# B&R Automation Studio project 2SegDemo (part 3)

#### WaveParFb.st
```iecst
(*
 This FB only atm works at 1ms cycle time

//Hz is times per second, in this case times is revolutions.
//To convert the Hz to revolutions and then scale by the task class cycle time
//1 hz, would mean that every TC cycle, we'd be incrementing by 2*PI/CycleTime

//Rx and Rz cylcic positions are always relative to the current position at the
//  ENABLING of the cyclic channel. Why? Who knows but that's the way it works
*)
FUNCTION_BLOCK WaveFb
	IF Enable AND Active AND Running THEN
		int.WaveCtrl.WaveX := int.WaveCtrl.WaveX + Pars.Wave.Freq / 1000 * 2 * 3.14;
		int.SlideCtrl.WaveX := int.SlideCtrl.WaveX + Pars.Slide.Freq / 1000 * 2 * 3.14;
		IF int.WaveCtrl.WaveX > 2 * 3.14 THEN
			int.WaveCtrl.WaveX := 0;
		END_IF

		IF int.SlideCtrl.WaveX > 2 * 3.14 THEN
			int.SlideCtrl.WaveX := 0;
		END_IF

		int.WaveCtrl.WaveY := SIN(int.WaveCtrl.WaveX);
		int.WaveCtrl.Height := int.WaveCtrl.WaveY * Pars.Wave.Amp + Pars.Wave.Center;

		//For the angle,just going to scale between -20/+20mRad.
		int.WaveCtrl.Angle := COS(int.WaveCtrl.WaveX) * 20;

		int.SlideCtrl.Height := SIN(int.SlideCtrl.WaveX) * 180 + 240;
	END_IF
	CASE int.State OF
		WAVE_IDLE: //**************************************************************** Idle State
			IF Enable THEN
				int.Fbs.GroupCreateFb.Controller := ADR(Controller);
				int.Fbs.GroupCreateFb.GroupID := 1;
				int.Fbs.GroupCreateFb.NumberOfShuttles := 2;
				int.Fbs.GroupCreateFb.ShuttleID[0] := 1;
				int.Fbs.GroupCreateFb.ShuttleID[1] := 2;
				int.Fbs.GroupCreateFb.Execute := TRUE;

				Active := TRUE;

				int.State := WAVE_CREATE_GROUP;
			END_IF
		WAVE_CREATE_GROUP: //**************************************************************** Create Sh Group
			IF int.Fbs.GroupCreateFb.Error THEN
				int.ErrorState := int.State;
				Error := TRUE;
				int.State := WAVE_ERROR;
			ELSIF int.Fbs.GroupCreateFb.Done THEN
				int.Fbs.GroupCreateFb.Execute := FALSE;

				int.Fbs.GroupCtrlFb.Controller := ADR(Controller);
				int.Fbs.GroupCtrlFb.CoupleMode := mcACP6D_GROUP_COUPLE_ONLY_XY;
				int.Fbs.GroupCtrlFb.GroupID := 1;
				int.Fbs.GroupCtrlFb.Option := mcACP6D_GROUP_COUPLE;
				int.Fbs.GroupCtrlFb.Execute := TRUE;

				int.State := WAVE_BOND_GROUP;
			END_IF
		WAVE_BOND_GROUP: //**************************************************************** Bond Sh Group
			IF int.Fbs.GroupCtrlFb.Error THEN
				int.ErrorState := int.State;
				Error := TRUE;
				int.State := WAVE_ERROR;
			ELSIF int.Fbs.GroupCtrlFb.Done THEN
				int.Fbs.GroupCtrlFb.Execute := FALSE;

				int.Fbs.ShortAxisFb.Controller := ADR(Controller);
				int.Fbs.ShortAxisFb.ShuttleID := 1; //Hard coded to 1 for now
				int.Fbs.ShortAxisFb.PositionZ := (Pars.Wave.Amp + Pars.Wave.Center) / 1000.0;
				int.Fbs.ShortAxisFb.PositionRx := 0.0;
				int.Fbs.ShortAxisFb.PositionRy := 0;
				int.Fbs.ShortAxisFb.PositionRz := 0;
				int.Fbs.ShortAxisFb.VelocityZ := 1;
				int.Fbs.ShortAxisFb.VelocityRx := 1;
				int.Fbs.ShortAxisFb.VelocityRy := 1;
				int.Fbs.ShortAxisFb.VelocityRz := 1;
				int.Fbs.ShortAxisFb.Execute := TRUE;

				int.State := WAVE_CFG_CHANNEL;
			END_IF
		WAVE_CFG_CHANNEL: //**************************************************************** Configure cyclic channel
			IF int.Fbs.ShortAxisFb.Error THEN
				int.ErrorState := int.State;
				Error := TRUE;
				int.State := WAVE_ERROR;
			ELSIF int.Fbs.ShortAxisFb.Done THEN
				int.Fbs.ShortAxisFb.Execute := FALSE;

				//Start at the peak of the sine wave, so pi/2
				int.WaveCtrl.WaveX := 1.57;
				int.SlideCtrl.WaveX := 1.57;
				int.WaveCtrl.WaveY := SIN(int.WaveCtrl.WaveX);
				int.WaveCtrl.Height := int.WaveCtrl.WaveY * Pars.Wave.Amp + Pars.Wave.Center;

				//For the angle,just going to scale between -25/+25mRad.
				int.WaveCtrl.Angle := COS(int.WaveCtrl.WaveX) * 25;

				int.Fbs.CyclicZFb.AxisID := 3;
				int.Fbs.CyclicZFb.ChannelID := 1;
				int.Fbs.CyclicZFb.Controller := ADR(Controller);
				int.Fbs.CyclicZFb.Value := (Pars.Wave.Amp + Pars.Wave.Center) - int.WaveCtrl.Height;
				int.Fbs.CyclicZFb.Enable := TRUE;

				int.Fbs.CyclicRxFb.AxisID := 5;
				int.Fbs.CyclicRxFb.ChannelID := 1;
				int.Fbs.CyclicRxFb.Controller := ADR(Controller);
				int.Fbs.CyclicRxFb.Value := 0;
				int.Fbs.CyclicRxFb.Enable := TRUE;

				int.Fbs.CyclicXFb.AxisID := 1;
				int.Fbs.CyclicXFb.ChannelID := 1;
				int.Fbs.CyclicXFb.Controller := ADR(Controller);
				int.Fbs.CyclicXFb.Value := 0.42;
				int.Fbs.CyclicXFb.Enable := TRUE;
				int.State := WAVE_SET_HEIGHT;
			END_IF

		WAVE_SET_HEIGHT: //**************************************************************** Set the starting height
			int.Fbs.CyclicChCtrlFb.Controller := ADR(Controller);
			int.Fbs.CyclicChCtrlFb.ShuttleID[0] := 1;
			int.Fbs.CyclicChCtrlFb.ChannelID[0] := 1;
			int.Fbs.CyclicChCtrlFb.AxisID[0].0 := TRUE; //X
			int.Fbs.CyclicChCtrlFb.AxisID[0].2 := TRUE; //Z
			int.Fbs.CyclicChCtrlFb.AxisID[0].4 := TRUE; //Ry
			int.Fbs.CyclicChCtrlFb.Execute := TRUE;
			int.Fbs.CyclicChCtrlFb.NumberOfShuttles := 1;
			int.Fbs.CyclicChCtrlFb.Level := 1;

			IF int.Fbs.CyclicChCtrlFb.Error THEN
				int.ErrorState := int.State;
				Error := TRUE;
				int.State := WAVE_ERROR;
			ELSIF int.Fbs.CyclicChCtrlFb.Done THEN
				int.Fbs.CyclicChCtrlFb.Execute := FALSE;
				Running := TRUE;
				int.State := WAVE_WAVE;
			END_IF
		WAVE_WAVE: //**************************************************************** Write channels, ride the wave
			int.Fbs.CyclicZFb.Value := -((Pars.Wave.Amp + Pars.Wave.Center) - int.WaveCtrl.Height) / 1000.0;
			int.Fbs.CyclicRxFb.Value := int.WaveCtrl.Angle / 1000.0;
			int.Fbs.CyclicXFb.Value := int.SlideCtrl.Height / 1000.0;

			IF NOT Enable THEN
				Running := FALSE;
				int.Fbs.CyclicZFb.Enable := FALSE;
				int.Fbs.CyclicRxFb.Enable := FALSE;
				int.Fbs.CyclicXFb.Enable := FALSE;
				int.Fbs.CyclicChCtrlFb.Execute := TRUE;
				int.Fbs.CyclicChCtrlFb.Level := 0;

				int.State := WAVE_EXIT_CFG;
			END_IF
		WAVE_EXIT_CFG:  //**************************************************************** Exit config channel
			IF int.Fbs.CyclicChCtrlFb.Error THEN
				int.ErrorState := int.State;
				Error := TRUE;
				int.State := WAVE_ERROR;
			ELSIF int.Fbs.CyclicChCtrlFb.Done THEN
				int.Fbs.CyclicChCtrlFb.Execute := FALSE;

				int.Fbs.ShortAxisFb.Controller := ADR(Controller);
				int.Fbs.ShortAxisFb.ShuttleID := 1;
				int.Fbs.ShortAxisFb.PositionZ := Pars.DefaultLevitationHeight;
				int.Fbs.ShortAxisFb.PositionRx := 0.0;
				int.Fbs.ShortAxisFb.PositionRy := 0;
				int.Fbs.ShortAxisFb.PositionRz := 0;
				int.Fbs.ShortAxisFb.VelocityZ := 1;
				int.Fbs.ShortAxisFb.VelocityRx := 1;
				int.Fbs.ShortAxisFb.VelocityRy := 1;
				int.Fbs.ShortAxisFb.VelocityRz := 1;
				int.Fbs.ShortAxisFb.Execute := TRUE;

				int.State := WAVE_MOVE_BACK;
			END_IF
		WAVE_MOVE_BACK: //**************************************************************** Move Back to level
			IF int.Fbs.ShortAxisFb.Error THEN
				int.ErrorState := int.State;
				Error := TRUE;
				int.State := WAVE_ERROR;
			ELSIF int.Fbs.ShortAxisFb.Done THEN
				int.Fbs.ShortAxisFb.Execute := FALSE;

				int.Fbs.GroupCtrlFb.Option := mcACP6D_GROUP_DECOUPLE;
				int.Fbs.GroupCtrlFb.Execute := TRUE;

				int.State := WAVE_UNBOUND_GROUP;
			END_IF
		WAVE_UNBOUND_GROUP: //**************************************************************** Unbond Sh Group
			IF int.Fbs.GroupCtrlFb.Error THEN
				int.ErrorState := int.State;
				Error := TRUE;
				int.State := WAVE_ERROR;
			ELSIF int.Fbs.GroupCtrlFb.Done THEN
				int.Fbs.GroupCtrlFb.Execute := FALSE;

				int.Fbs.GroupDeleteFb.Controller := ADR(Controller);
				int.Fbs.GroupDeleteFb.GroupID := 1;
				int.Fbs.GroupDeleteFb.Execute := TRUE;

				int.State := WAVE_DELETE_GROUP;
			END_IF
		WAVE_DELETE_GROUP: //**************************************************************** Delete Sh Group
			IF int.Fbs.GroupDeleteFb.Error THEN
				int.ErrorState := int.State;
				Error := TRUE;
				int.State := WAVE_ERROR;
			ELSIF int.Fbs.GroupDeleteFb.Done THEN
				int.Fbs.GroupDeleteFb.Execute := FALSE;

				Active := FALSE;
				int.WaveCtrl.WaveX := 0;
				int.SlideCtrl.WaveX := 0;
				int.State := WAVE_IDLE;
			END_IF
		WAVE_ERROR: //**************************************************************** Error State
			IF NOT Enable THEN

				Active := FALSE;
				Error := FALSE;
				Running := FALSE;

				int.Fbs.ShortAxisFb.Execute := FALSE;
				int.Fbs.CyclicChCtrlFb.Execute := FALSE;
				int.Fbs.CyclicZFb.Enable := FALSE;
				int.Fbs.CyclicRxFb.Enable := FALSE;
				int.Fbs.CyclicXFb.Enable := FALSE;
				int.Fbs.GroupCreateFb.Execute := FALSE;
				int.Fbs.GroupCtrlFb.Execute := FALSE;
				int.Fbs.GroupDeleteFb.Execute := FALSE;

				int.WaveCtrl.WaveX := 0;
				int.SlideCtrl.WaveX := 0;
				int.State := WAVE_IDLE;
			END_IF

	END_CASE;

	int.Fbs.ShortAxisFb();
	int.Fbs.CyclicChCtrlFb();
	int.Fbs.CyclicZFb();
	int.Fbs.CyclicRxFb();
	int.Fbs.CyclicXFb();
	int.Fbs.GroupCreateFb();
	int.Fbs.GroupCtrlFb();
	int.Fbs.GroupDeleteFb();

END_FUNCTION_BLOCK
```

#### AntiSloshFb.st
```iecst
FUNCTION_BLOCK AntiSloshFb

END_FUNCTION_BLOCK
```

#### LandFb.st
```iecst
FUNCTION_BLOCK LandFb

	CASE int.State OF
		LAND_IDLE: //**************************************************************** Idle State
			IF Enable THEN
				Active := TRUE;

				int.State := LAND_WAIT;
			END_IF
		LAND_ISSUE_CMD: //**************************************************************** Create Sh Group
			IF int.Fbs.LandFb.Error THEN
				int.ErrorState := int.State;
				Error := TRUE;
				int.State := LAND_ERROR;
			ELSIF NOT Enable AND int.Fbs.LandFb.Done THEN
				int.Fbs.LandFb.Execute := FALSE;

				int.State := LAND_RESET;
			ELSIF int.Fbs.LandFb.Done THEN
				int.Landed := NOT int.Landed;
				int.Fbs.LandFb.Execute := FALSE;

				int.State := LAND_WAIT;
			END_IF
		LAND_WAIT: //**************************************************************** Waiting for an update cmd
			IF NOT Enable THEN
				IF Land THEN
					int.Fbs.LandFb.Controller := ADR(Controller);
					int.Fbs.LandFb.Level := mcACP6D_LEVEL_LEVITATE;
					int.Fbs.LandFb.ShuttleID := Pars.ShId;
					int.Fbs.LandFb.Execute := TRUE;

					int.State := LAND_ISSUE_CMD;
				ELSE
					int.State := LAND_RESET;
				END_IF
			ELSIF (Land AND NOT int.Landed) OR (NOT Land AND int.Landed) THEN
				IF int.Landed THEN
					int.Fbs.LandFb.Level := mcACP6D_LEVEL_LEVITATE;
				ELSE
					int.Fbs.LandFb.Level := mcACP6D_LEVEL_LAND;
				END_IF
				int.Fbs.LandFb.Controller := ADR(Controller);
				int.Fbs.LandFb.ShuttleID := Pars.ShId;
				int.Fbs.LandFb.Execute := TRUE;

				int.State := LAND_ISSUE_CMD;
			END_IF

		LAND_ERROR: //**************************************************************** Error STate
			IF NOT Enable THEN
				int.State := LAND_RESET;
			END_IF

		LAND_RESET: //**************************************************************** Reset state
			Active := FALSE;
			Error := FALSE;
			int.Landed := FALSE;

			int.Fbs.LandFb.Execute := FALSE;

			int.State := LAND_IDLE;
	END_CASE;

	int.Fbs.LandFb();
END_FUNCTION_BLOCK
```

#### GenericDemoFb.st
```iecst
FUNCTION_BLOCK GenericMotionDemoFB

	CASE int.State OF
		GEN_IDLE: //**************************************************************** Idle State
			IF Enable THEN
				Active := TRUE;

				int.Fbs.BufferCtrl.Controller := ADR(Controller);
				int.Fbs.BufferCtrl.Option := mcACP6D_BUFFER_BLOCK;
				int.Fbs.BufferCtrl.ShuttleID := 0;
				int.Fbs.BufferCtrl.Execute := TRUE;

				int.State := GEN_BLOCK_BUFFER;
			END_IF
		GEN_BLOCK_BUFFER: //**************************************************************** Block Buffer
			IF int.Fbs.BufferCtrl.Error THEN
				int.ErrorState := int.State;
				Error := TRUE;
				int.State := GEN_ERROR;
			ELSIF int.Fbs.BufferCtrl.Done THEN
				int.Fbs.BufferCtrl.Execute := FALSE;

				int.Fbs.MacroRunFB.Controller := ADR(Controller);
				int.Fbs.MacroRunFB.ShuttleID := Pars.ShId[0];
				int.Fbs.MacroRunFB.MacroID := Pars.MacroId[0];
				int.Fbs.MacroRunFB.Execute := TRUE;

				int.State := GEN_RUN_MACRO1;
			END_IF
		GEN_RUN_MACRO1: //**************************************************************** Run Macro 1
			IF int.Fbs.MacroRunFB.Error THEN
				int.ErrorState := int.State;
				Error := TRUE;
				int.State := GEN_ERROR;
			ELSIF int.Fbs.MacroRunFB.Acknowledge THEN
				int.Fbs.MacroRunFB.Execute := FALSE;
				int.Fbs.MacroRunFB.ShuttleID := Pars.ShId[1];
				int.Fbs.MacroRunFB.MacroID := Pars.MacroId[1];

				int.State := GEN_RUN_MACRO2;
			END_IF
		GEN_RUN_MACRO2: //**************************************************************** Run Macro 2
			int.Fbs.MacroRunFB.Execute := TRUE;
			IF int.Fbs.MacroRunFB.Error THEN
				int.ErrorState := int.State;
				Error := TRUE;
				int.State := GEN_ERROR;
			ELSIF int.Fbs.MacroRunFB.Acknowledge THEN
				int.Fbs.MacroRunFB.Execute := FALSE;

				int.Fbs.BufferCtrl.Option := mcACP6D_BUFFER_RELEASE;
				int.Fbs.BufferCtrl.Execute := TRUE;

				int.State := GEN_RELEASE_BUFFER;
			END_IF

		GEN_RELEASE_BUFFER: //**************************************************************** Block Buffer
			IF int.Fbs.BufferCtrl.Error THEN
				int.ErrorState := int.State;
				Error := TRUE;
				int.State := GEN_ERROR;
			ELSIF int.Fbs.BufferCtrl.Done THEN
				int.Fbs.BufferCtrl.Execute := FALSE;

				int.State := GEN_RUN_DEMO;
			END_IF
		GEN_RUN_DEMO: //**************************************************************** Run Demo State
			IF NOT Enable THEN
				int.Fbs.StopFb.Controller := ADR(Controller);
				int.Fbs.StopFb.ShuttleID := 0;
				int.Fbs.StopFb.Execute := TRUE;
				int.State := GEN_STOP;
			END_IF
		GEN_STOP:  //**************************************************************** Stopping Shuttle state
			IF int.Fbs.StopFb.Error THEN
				int.ErrorState := int.State;
				Error := TRUE;
				int.State := GEN_ERROR;
			ELSIF int.Fbs.StopFb.Done THEN
				int.Fbs.StopFb.Execute := FALSE;

				int.Fbs.ShortAxisFb.Controller := ADR(Controller);
				int.Fbs.ShortAxisFb.PositionZ := 0.001;
				int.Fbs.ShortAxisFb.ShuttleID := Pars.ShId[0];
				int.Fbs.ShortAxisFb.VelocityZ := 1;
				int.Fbs.ShortAxisFb.Execute := TRUE;

				int.State := GEN_RESET_HEIGHT1;
			END_IF
		GEN_RESET_HEIGHT1: //**************************************************************** Reset Height 1
			IF int.Fbs.ShortAxisFb.Error THEN
				int.ErrorState := int.State;
				Error := TRUE;
				int.State := GEN_ERROR;
			ELSIF int.Fbs.ShortAxisFb.Done THEN
				int.Fbs.ShortAxisFb.Execute := FALSE;

				int.Fbs.ShortAxisFb.ShuttleID := Pars.ShId[1];
				int.State := GEN_RESET_HEIGHT2;
			END_IF
		GEN_RESET_HEIGHT2: //**************************************************************** Reset Height 2
			int.Fbs.ShortAxisFb.Execute := TRUE;
			IF int.Fbs.ShortAxisFb.Error THEN
				int.ErrorState := int.State;
				Error := TRUE;
				int.State := GEN_ERROR;
			ELSIF int.Fbs.ShortAxisFb.Done THEN
				int.Fbs.ShortAxisFb.Execute := FALSE;

				int.State := GEN_RESET;
			END_IF
		GEN_ERROR: //**************************************************************** Error state
			IF NOT Enable THEN
				int.State := GEN_RESET;
			END_IF

		GEN_RESET: //**************************************************************** Reset state
			Active := FALSE;
			Error := FALSE;

			int.Fbs.ShortAxisFb.Execute := FALSE;
			int.Fbs.BufferCtrl.Execute := FALSE;
			int.Fbs.MacroRunFB.Execute := FALSE;
			int.Fbs.StopFb.Execute := FALSE;

			int.State := GEN_IDLE;;
	END_CASE;

	int.Fbs.ShortAxisFb();
	int.Fbs.BufferCtrl();
	int.Fbs.MacroRunFB();
	int.Fbs.StopFb();

END_FUNCTION_BLOCK
```

### Program Logical/Source/Demos/MixDemo

#### Types.typ
```iecst
TYPE
	MoveTyp : 	STRUCT
		X : REAL;
		Y : REAL;
		Vel : REAL;
		Accel : REAL;
		EndVel : REAL;
		Angle : REAL;
	END_STRUCT;
	FbsTyp : 	STRUCT
		MovePlaneFb : MC_BR_MoveInPlane_Acp6D;
		MoveArcFb : MC_BR_MoveArcAngle_Acp6D;
		Wait : TON;
		RunMacroFb : MC_BR_MacroRun_Acp6D;
		LoadMacroFb : MC_BR_MacroLoad_Acp6D;
	END_STRUCT;
END_TYPE
```

#### Variables.var
```iecst
VAR
	Fbs : FbsTyp;
	state : UDINT;
	shId : USINT;
END_VAR
VAR RETAIN
	run : BOOL;
END_VAR
VAR
	macroId : USINT;
END_VAR
```

#### Cyclic.st
```iecst
//Mixing demo

(*
	Move shuttle to segment center position
	Wait for some time (here food coloring is added)
	Preform mixing movement
	Move back to other side
	Wait for some time (food coloring added)
	Preform mixing movement
	Move shuttle to start position

*)

PROGRAM _CYCLIC
	Fbs.LoadMacroFb.Controller := ADR(gMcAcp6DController);

	Fbs.RunMacroFb.Controller := ADR(gMcAcp6DController);
	Fbs.RunMacroFb.ShuttleID := shId;
	Fbs.RunMacroFb.MacroID := macroId;

	CASE state OF
		0:
			Fbs.LoadMacroFb.MacroID := macroId;
			IF run THEN
				Fbs.RunMacroFb.Execute := TRUE;
				Fbs.RunMacroFb.MacroID := 130;
				state := 10;
			END_IF
		10:
			IF Fbs.RunMacroFb.Done THEN
				Fbs.RunMacroFb.Execute := FALSE;
				state := 11;
			END_IF
		11:
			Fbs.RunMacroFb.Execute := TRUE;
			Fbs.RunMacroFb.MacroID := 131;
			state := 20;
		20:
			IF Fbs.RunMacroFb.Done THEN
				Fbs.RunMacroFb.Execute := FALSE;
				state := 21;
			END_IF
		21:
			Fbs.RunMacroFb.Execute := TRUE;
			Fbs.RunMacroFb.MacroID := 132;
			state := 30;
		30:
			IF Fbs.RunMacroFb.Done THEN
				Fbs.RunMacroFb.Execute := FALSE;
				state := 31;
			END_IF
		31:
			Fbs.RunMacroFb.Execute := TRUE;
			Fbs.RunMacroFb.MacroID := 131;
			state := 40;
		40:
			IF Fbs.RunMacroFb.Done THEN
				Fbs.RunMacroFb.Execute := FALSE;

				Fbs.MovePlaneFb.Controller := ADR(gMcAcp6DController);
				Fbs.MovePlaneFb.ShuttleID := shId;
				Fbs.MovePlaneFb.PositionX := 0.24;
				Fbs.MovePlaneFb.PositionY := 0.12;
				Fbs.MovePlaneFb.Velocity := 0.5;
				Fbs.MovePlaneFb.Acceleration := 1;
				Fbs.MovePlaneFb.Execute := TRUE;
				state := 50;
			END_IF
		50:
			IF Fbs.MovePlaneFb.Done THEN
				Fbs.MovePlaneFb.Execute := FALSE;
				run := FALSE;
				state := 0;
			END_IF
	END_CASE;

	Fbs.LoadMacroFb();
	Fbs.MovePlaneFb();
	Fbs.RunMacroFb();
END_PROGRAM
```

#### Init.st
```iecst
PROGRAM _INIT
	Fbs.LoadMacroFb.FileDevice := '6DMacro';
	Fbs.LoadMacroFb.FileName := '130_MixDemo.xml';
	macroId := 130;
	shId := 1;
END_PROGRAM
```

### Package Logical/Source/Main - Package that contains the main entry point to the machine

### Program Logical/Source/Main/Main

#### Types.typ
```iecst
TYPE
	MainFbsTyp : 	STRUCT
		TimerFb : TON;
		StopAllFb : MC_BR_Stop_Acp6D;
	END_STRUCT;
	MainStatesEnum :
		(
		MAIN_OFF,
		MAIN_INIT,
		MAIN_RECOVERING,
		MAIN_READY,
		MAIN_STARTING,
		MAIN_RUN_PROCESS,
		MAIN_RUN_DANCE,
		MAIN_STOPPING,
		MAIN_ERROR,
		MAIN_RESET
		);
END_TYPE
```

#### Variables.var
```iecst
VAR
	i : USINT; (*Loop index*)
	state : MainStatesEnum; (*State of system*)
	Fbs : MainFbsTyp;
END_VAR
```

#### Cyclic.st
```iecst
PROGRAM _CYCLIC
	IF gAcp6DCtrlIf.Sts.Error THEN
		state := MAIN_ERROR;
	END_IF

	IF gMainIf.Cmd.StopAllShuttles THEN
		Fbs.StopAllFb.Controller := ADR(gMcAcp6DController);
		Fbs.StopAllFb.Execute := TRUE;
		IF Fbs.StopAllFb.Done OR Fbs.StopAllFb.Error THEN
			Fbs.StopAllFb.Execute := FALSE;
			gMainIf.Cmd.StopAllShuttles := FALSE;
		END_IF
	END_IF

	CASE state OF
		MAIN_OFF: //******************************************************************************** Main Off State
			IF gMainIf.Cmd.Power THEN
				gAcp6DCtrlIf.Cmd.Power := gMainIf.Cfg.Enable6D;

				state := MAIN_INIT;
			END_IF

		MAIN_INIT: //******************************************************************************** Main Initializing State
			IF (gAcp6DCtrlIf.Sts.PowerOn AND gAcp6DCtrlIf.Sts.Ready OR NOT gMainIf.Cfg.Enable6D) THEN
				gMainIf.Sts.Power6D := TRUE;

				state := MAIN_READY;
			ELSIF NOT gMainIf.Cmd.Power THEN
				gAcp6DCtrlIf.Cmd.Power := FALSE;

				gMainIf.Sts.Power6D := FALSE;

				state := MAIN_OFF;
			END_IF
		MAIN_RECOVERING: //******************************************************************************** Main Recovery State
			IF (g6DRecoveryIf.Sts.ReadyToStartProc OR NOT gMainIf.Cfg.Enable6D) THEN
				g6DRecoveryIf.Cmd.Recover := FALSE;

				state := MAIN_READY;
			END_IF
		MAIN_READY://******************************************************************************** Main Ready State
			IF NOT gMainIf.Cmd.Power THEN
				gMainIf.Sts.Power6D := FALSE;
				gAcp6DCtrlIf.Cmd.Power := FALSE;

				state := MAIN_OFF;
			END_IF

		MAIN_STARTING://******************************************************************************** Main Starting State
			IF gAcp6DCtrlIf.Sts.Error THEN
				state := MAIN_ERROR;
			ELSIF NOT gMainIf.Cmd.Power THEN
				gMainIf.Cmd.StartDemoCycle := FALSE;
				gMainIf.Sts.Power6D := FALSE;
				gAcp6DCtrlIf.Cmd.Power := FALSE;

				state := MAIN_OFF;
			END_IF

		MAIN_RUN_PROCESS: //******************************************************************************** Main Process State
		MAIN_STOPPING: //******************************************************************************** Main Stopping State

		MAIN_ERROR: //******************************************************************************** Main Error State
			IF gMainIf.Cmd.Reset THEN
				gMainIf.Cmd.Reset := FALSE;

				gMainIf.Sts.Running := FALSE;
				gAcp6DCtrlIf.Cmd.ErrorReset := TRUE;
				Fbs.TimerFb.IN := FALSE;

				IF gMainIf.Cmd.Power THEN
					state := MAIN_READY;
				ELSE
					state := MAIN_OFF;
				END_IF
			END_IF
	END_CASE;

	Fbs.StopAllFb();
END_PROGRAM
```

#### Init.st
```iecst
PROGRAM _INIT
	gMainIf.Cfg.ShuttleCount := 8;

	gMainIf.Cfg.Enable6D := TRUE;
	gMainIf.Cfg.EnableRobot := TRUE;

	gMainIf.Par.ProcessDemoTime := T#120s;
	gMainIf.Par.DanceDemoTime := T#180s;

	//Used to initialize the shuttle indecies.
	FOR i:=0 TO gMainIf.Cfg.ShuttleCount-1 DO
		gShuttleIf[i].Cfg.ShuttleId := i + 1;
	END_FOR;

END_PROGRAM
```

### Package Logical/Source/6DCtrl - Package containing the main logic for controlling the 6D system as a whole

### Acp6DTypes.typ
```iecst
(*Datatypes for the Load Macro Interface*)

TYPE
	gMacroLoadIfTYp : 	STRUCT
		Cmd : gMacroLoadIfCmdTyp;
		Par : gMacroLoadIfParTyp;
		Sts : gMacroLoadIfStatusTyp;
	END_STRUCT;
	gMacroLoadIfCmdTyp : 	STRUCT
		LoadAll : BOOL; (*Command to load all macros*)
		Clear : BOOL; (*Command to clear a singular macro*)
		LoadSingle : BOOL; (*Commadn to load a singular macro*)
		Reset : BOOL; (*Command to reset the macro load interface. Also resets the "AllMacroLoaded" status*)
	END_STRUCT;
	MacroParTyp : 	STRUCT
		Load : BOOL; (*Flag To denote that we should load the macro*)
		MacroFileName : STRING[80]; (*XML File Name of the Macro to load*)
		MacroID : USINT; (*MacroID of the associated macro*)
	END_STRUCT;
	gMacroLoadIfParTyp : 	STRUCT
		FileDevice : STRING[80]; (*FileDevice to find the macro *)
		MacroList : ARRAY[0..MAX_MACRO_COUNT_ARRAY]OF MacroParTyp; (*List of macros to load*)
		SingleMacroLoad : MacroParTyp; (*Parameter to load a singular macro*)
	END_STRUCT;
	gMacroLoadIfStatusTyp : 	STRUCT
		AllMacrosLoaded : BOOL;
		Loading : BOOL;
		CurrentMacro : USINT;
		CmdDone : BOOL;
		Error : BOOL;
		MacroIDError : USINT;
	END_STRUCT;
END_TYPE
```

### Program Logical/Source/6DCtrl/6DCtrl (IEC)

#### Cyclic.st
```iecst
PROGRAM _CYCLIC

	IF((Fbs.SysReadStateFb.Valid AND Fbs.SysReadStateFb.State = mcACP6D_STATE_ERROR) AND (state <> ACP6D_ERROR))THEN
		state := ACP6D_ERROR;
	END_IF;

	CASE state OF
		ACP6D_RESET: 	//******************************************************************************** 6D Reset State
			IF(Fbs.SysReadStateFb.Valid AND (Fbs.SysReadStateFb.State = mcACP6D_STATE_INACTIVE))THEN
				state := ACP6D_INACTIVE;
			ELSIF(Fbs.SysReadStateFb.State = mcACP6D_STATE_OPERATION)THEN
				state := ACP6D_POWER_OFF;
			END_IF;

		ACP6D_POWER_OFF: 	//******************************************************************************** 6D Power off commanding State
			Fbs.PowerOffFb.Execute := TRUE;
			IF(Fbs.PowerOffFb.Acknowledge AND (Fbs.SysReadStateFb.Valid AND Fbs.SysReadStateFb.State = mcACP6D_STATE_INACTIVE))THEN
				gAcp6DCtrlIf.Sts.PowerOn := FALSE;
				Fbs.PowerOffFb.Execute 	:= FALSE;
				state := ACP6D_INACTIVE;
			ELSIF(Fbs.PowerOffFb.Error)THEN
				Fbs.PowerOffFb.Execute 	:= FALSE;
				gAcp6DCtrlIf.Sts.ErrorID := Fbs.PowerOffFb.ErrorID;
				state := ACP6D_ERROR;
			END_IF;

		ACP6D_INACTIVE:	 	//******************************************************************************** 6D Inactive/Power Off state
			IF(gAcp6DCtrlIf.Cmd.Power)THEN
				Fbs.PowerOnFb.Execute := TRUE;
				//MpAuditCustomEvent(gAuditTrail,"INFO","Acp6DSys","Power On Command Issued");
				state := ACP6D_POWER_ON;
			END_IF;

		ACP6D_POWER_ON: 	//******************************************************************************** 6D Power on Commanding State
			IF Fbs.PowerOnFb.Error THEN
				gAcp6DCtrlIf.Sts.ErrorID := Fbs.PowerOnFb.ErrorID;
				state := ACP6D_ERROR;
			ELSIF(Fbs.PowerOnFb.Acknowledge AND (Fbs.SysReadStateFb.Valid AND (Fbs.SysReadStateFb.State > mcACP6D_STATE_INACTIVE)))THEN
				//MpAuditCustomEvent(gAuditTrail,"INFO","Acp6DSys","Powered On");
				Fbs.PowerOnFb.Execute := FALSE;
				state := ACP6D_WAIT_ACTIVATION;
			END_IF;

			//Necessary state when using Absolute ID.
		ACP6D_WAIT_ACTIVATION: 	//******************************************************************************** 6D Waiting for Activation of Shuttles State
			IF(Fbs.SysReadStateFb.Valid)THEN
				IF(Fbs.SysReadStateFb.State = mcACP6D_STATE_OPERATION)THEN
					gAcp6DCtrlIf.Sts.PowerOn := TRUE;
					IF gAcp6DCtrlIf.Par.MacroEnabled THEN

						state := ACP6D_INIT_MACRO;
					ELSE
						state := ACP6D_READY;
					END_IF
				ELSIF(Fbs.SysReadStateFb.State = mcACP6D_STATE_INACTIVE)THEN
					state := ACP6D_INACTIVE; // Error during Activating state; Can happen in Absolute ID mode.
					gAcp6DCtrlIf.Cmd.Power := FALSE;
				END_IF;
			END_IF;
		ACP6D_INIT_MACRO: 	//******************************************************************************** 6D Wait for Macro initilization State
			IF gMacroLoadIf.Sts.AllMacrosLoaded THEN
				gMacroLoadIf.Cmd.LoadAll := FALSE;

				state := ACP6D_READY;
			ELSE
				gMacroLoadIf.Cmd.LoadAll := TRUE;
			END_IF
		ACP6D_CFG_CYCLIC_CHANNEL: 	//******************************************************************************** 6D Confiugring the cyclic channel reads
			IF Fbs.CfgReadCyclicPos.Error THEN
				gAcp6DCtrlIf.Sts.Error := TRUE;
				gAcp6DCtrlIf.Sts.ErrorID := Fbs.CfgReadCyclicPos.ErrorID;

				state := ACP6D_ERROR;
			ELSIF Fbs.CfgReadCyclicPos.Done THEN
				Fbs.CfgReadCyclicPos.Execute := FALSE;

				state := ACP6D_READY;
			END_IF
		ACP6D_READY: 	//******************************************************************************** 6D Ready/Running State
			IF(NOT gAcp6DCtrlIf.Cmd.Power)THEN
				gMacroLoadIf.Cmd.Reset := TRUE;
				state := ACP6D_POWER_OFF;
			END_IF;

		ACP6D_ERROR: 	//******************************************************************************** 6D Error State
			gAcp6DCtrlIf.Sts.PowerOn := FALSE;
			IF(gAcp6DCtrlIf.Cmd.ErrorReset)THEN
				IF(Fbs.SysReadStateFb.State<>mcACP6D_STATE_ERROR)THEN
					gAcp6DCtrlIf.Cmd.ErrorReset := FALSE;
					state := ACP6D_RESET;
				ELSE
					Fbs.PowerOffFb.Execute := TRUE;	 // Reset error with power off.
					IF(Fbs.PowerOffFb.Acknowledge)THEN
						gMacroLoadIf.Cmd.Reset := TRUE;
						Fbs.PowerOffFb.Execute 	:= FALSE;
					ELSIF(Fbs.PowerOffFb.Error)THEN
						gAcp6DCtrlIf.Cmd.ErrorReset := FALSE;
						Fbs.PowerOffFb.Execute 	:= FALSE;
						gAcp6DCtrlIf.Sts.ErrorID := Fbs.PowerOffFb.ErrorID;
						state := ACP6D_ERROR;
					END_IF;
				END_IF;
			END_IF;
	END_CASE;

	FOR i:=0 TO gMainIf.Cfg.ShuttleCount - 1 DO
		Fbs.ShReadPositionFb[i].Controller := ADR(gMcAcp6DController);
		Fbs.ShReadPositionFb[i].Enable := TRUE;
		Fbs.ShReadPositionFb[i].ShuttleID := gShuttleIf[i].Cfg.ShuttleId;
		Fbs.ShReadPositionFb[i]();

		Fbs.ShReadForceFb[i].Controller := ADR(gMcAcp6DController);
		Fbs.ShReadForceFb[i].Enable := TRUE;
		Fbs.ShReadForceFb[i].ShuttleID := gShuttleIf[i].Cfg.ShuttleId;
		Fbs.ShReadForceFb[i]();

		Fbs.ShReadState[i].Controller := ADR(gMcAcp6DController);
		Fbs.ShReadState[i].Enable := TRUE;
		Fbs.ShReadState[i].ShuttleID := gShuttleIf[i].Cfg.ShuttleId;
		Fbs.ShReadState[i]();

		gShuttleIf[i].Sts.ShuttleInfo.Force.Value := Fbs.ShReadForceFb[i].ForceInfo;
		gShuttleIf[i].Sts.ShuttleInfo.Force.Valid := Fbs.ShReadForceFb[i].Valid;
		gShuttleIf[i].Sts.ShuttleInfo.Position.Value := Fbs.ShReadPositionFb[i].PositionInfo;
		gShuttleIf[i].Sts.ShuttleInfo.Position.Valid := Fbs.ShReadPositionFb[i].Valid;
		gShuttleIf[i].Sts.ShuttleInfo.State.Value := Fbs.ShReadState[i].State;
		gShuttleIf[i].Sts.ShuttleInfo.State.Valid := Fbs.ShReadState[i].Valid;
	END_FOR;

	IF gAcp6DCtrlIf.Cmd.GetErrorInfo THEN
		Fbs.GetErrorCodesFb.Controller := ADR(gMcAcp6DController);
		Fbs.GetErrorCodesFb.Execute := TRUE;

		IF Fbs.GetErrorCodesFb.Valid OR Fbs.GetErrorCodesFb.Error THEN
			gAcp6DCtrlIf.Sts.ErrorCodes := Fbs.GetErrorCodesFb.ErrorCodes;
			Fbs.GetErrorCodesFb.Execute := FALSE;
			gAcp6DCtrlIf.Cmd.GetErrorInfo := FALSE;
		END_IF

	END_IF
	Fbs.CfgReadCyclicPos();
	Fbs.GetErrorCodesFb();
	Fbs.SysReadStateFb();
	Fbs.PowerOffFb();
	Fbs.PowerOnFb();
	Fbs.AutoRefreshFB();

	gAcp6DCtrlIf.Sts.Ready := state = ACP6D_READY;
	gAcp6DCtrlIf.Sts.Error := state = ACP6D_ERROR;
	gAcp6DCtrlIf.Sts.ReadyToPowerOn := Fbs.SysReadStateFb.Valid AND Fbs.SysReadStateFb.State = mcACP6D_STATE_INACTIVE;
END_PROGRAM
```

#### Init.st
```iecst
PROGRAM _INIT
	gMcAcp6DController.H2P_START := ADR(FBout);
	gMcAcp6DController.P2H_START := ADR(FBin);
	gMcAcp6DController.ConfiguredFeedbackStreamAxis	:= 63;

	Fbs.AutoRefreshFB.Controller	:= ADR(gMcAcp6DController);
	Fbs.PowerOffFb.Controller := ADR(gMcAcp6DController);
	Fbs.PowerOnFb.Controller := ADR(gMcAcp6DController);
	Fbs.SysReadStateFb.Controller := ADR(gMcAcp6DController);

	Fbs.AutoRefreshFB.Enable := TRUE;
	Fbs.SysReadStateFb.Enable := TRUE;

	gAcp6DCtrlIf.Par.MacroEnabled := TRUE;
END_PROGRAM
```

### Program Logical/Source/6DCtrl/MacroLoad (IEC)

#### Cyclic.st
```iecst
PROGRAM _CYCLIC
	CASE state OF
		MACLOAD_IDLE:	//******************************************************************************** Macro Idle State
			IF gMacroLoadIf.Cmd.LoadAll OR gMacroLoadIf.Cmd.LoadSingle THEN
				gMacroLoadIf.Sts.AllMacrosLoaded := FALSE;
				gMacroLoadIf.Sts.Loading := TRUE;
				gMacroLoadIf.Sts.CurrentMacro := 0;

				state := MACLOAD_COUNT_CHECK;
			ELSIF gMacroLoadIf.Cmd.Clear THEN
				MacroFbs.MacroClearFb.Controller := ADR(gMcAcp6DController);
				MacroFbs.MacroClearFb.MacroID := gMacroLoadIf.Par.SingleMacroLoad.MacroID;
				MacroFbs.MacroClearFb.Execute := TRUE;

				state := MACLOAD_CLEAR;
			ELSIF gMacroLoadIf.Cmd.Reset THEN
				gMacroLoadIf.Sts.AllMacrosLoaded := FALSE;
				gMacroLoadIf.Cmd.Reset := FALSE;
			END_IF

		MACLOAD_LOAD://******************************************************************************** Macro Load State
			IF MacroFbs.MacroLoadFb.Error THEN
				gMacroLoadIf.Sts.Error := TRUE;
				gMacroLoadIf.Sts.MacroIDError := gMacroLoadIf.Sts.CurrentMacro;

				state := MACLOAD_ERROR;
			ELSIF MacroFbs.MacroLoadFb.Done THEN
				MacroFbs.MacroLoadFb.Execute := FALSE;
				IF gMacroLoadIf.Cmd.LoadSingle THEN
					gMacroLoadIf.Cmd.LoadSingle := FALSE;
					gMacroLoadIf.Sts.CmdDone := TRUE;
					state := MACLOAD_DONE;
				ELSE //Means we commanded a "LOAD ALL"
					gMacroLoadIf.Sts.CurrentMacro := gMacroLoadIf.Sts.CurrentMacro + 1;

					state := MACLOAD_COUNT_CHECK;
				END_IF
			END_IF

		MACLOAD_COUNT_CHECK: //******************************************************************************** Macro Count check State
			IF gMacroLoadIf.Par.MacroList[gMacroLoadIf.Sts.CurrentMacro].Load THEN
				MacroFbs.MacroLoadFb.Controller := ADR(gMcAcp6DController);
				MacroFbs.MacroLoadFb.FileDevice := gMacroLoadIf.Par.FileDevice;
				IF gMacroLoadIf.Cmd.LoadAll THEN
					MacroFbs.MacroLoadFb.MacroID := gMacroLoadIf.Par.MacroList[gMacroLoadIf.Sts.CurrentMacro].MacroID;
					MacroFbs.MacroLoadFb.FileName := gMacroLoadIf.Par.MacroList[gMacroLoadIf.Sts.CurrentMacro].MacroFileName;

				ELSIF gMacroLoadIf.Cmd.LoadSingle THEN
					MacroFbs.MacroLoadFb.MacroID := gMacroLoadIf.Par.SingleMacroLoad.MacroID;
					MacroFbs.MacroLoadFb.FileName := gMacroLoadIf.Par.SingleMacroLoad.MacroFileName;
				END_IF
				MacroFbs.MacroLoadFb.Execute := TRUE;
				state := MACLOAD_LOAD;
			ELSE
				gMacroLoadIf.Sts.CurrentMacro := gMacroLoadIf.Sts.CurrentMacro + 1;
				IF gMacroLoadIf.Sts.CurrentMacro >= MAX_MACRO_COUNT THEN
					gMacroLoadIf.Sts.AllMacrosLoaded := TRUE;
					gMacroLoadIf.Sts.CmdDone := TRUE;

					state := MACLOAD_DONE;
				END_IF
			END_IF
		MACLOAD_CLEAR: //******************************************************************************** Macro Clear state
			IF MacroFbs.MacroClearFb.Error THEN
				gMacroLoadIf.Sts.Error := TRUE;

				state := MACLOAD_ERROR;
			ELSIF MacroFbs.MacroClearFb.Done THEN
				MacroFbs.MacroClearFb.Execute := FALSE;
				gMacroLoadIf.Sts.CmdDone := TRUE;

				state := MACLOAD_DONE;
			END_IF
		MACLOAD_DONE: //******************************************************************************** Load Done State
			gMacroLoadIf.Sts.Loading := FALSE;
			IF NOT gMacroLoadIf.Cmd.Clear AND NOT gMacroLoadIf.Cmd.LoadAll AND NOT gMacroLoadIf.Cmd.LoadSingle THEN
				gMacroLoadIf.Sts.CmdDone := FALSE;
				state := MACLOAD_IDLE;
			END_IF
		MACLOAD_ERROR: //******************************************************************************** Macro load error State
			IF gMacroLoadIf.Cmd.Reset THEN
				MacroFbs.MacroClearFb.Execute := FALSE;
				MacroFbs.MacroLoadFb.Execute := FALSE;

				gMacroLoadIf.Cmd.Reset := FALSE;

				gMacroLoadIf.Sts.Loading := FALSE;
				gMacroLoadIf.Sts.AllMacrosLoaded := FALSE;
				gMacroLoadIf.Sts.Error := FALSE;
				gMacroLoadIf.Sts.MacroIDError := 0;
				state := MACLOAD_IDLE;
			END_IF
	END_CASE;

	//FB Calls
	MacroFbs.MacroLoadFb();
	MacroFbs.MacroClearFb();
END_PROGRAM
```

#### Init.st
```iecst
PROGRAM _INIT
	gMacroLoadIf.Par.SingleMacroLoad.Load := TRUE;

		//Fill Station 2
	gMacroLoadIf.Par.MacroList[0].Load := TRUE;
	gMacroLoadIf.Par.MacroList[0].MacroFileName := '135_UpDown.xml';
	gMacroLoadIf.Par.MacroList[0].MacroID := 135;

	gMacroLoadIf.Par.MacroList[1].Load := TRUE;
	gMacroLoadIf.Par.MacroList[1].MacroFileName := '136_DownUp.xml';
	gMacroLoadIf.Par.MacroList[1].MacroID := 136;

	gMacroLoadIf.Par.MacroList[2].Load := TRUE;
	gMacroLoadIf.Par.MacroList[2].MacroFileName := '137_LevUpDown.xml';
	gMacroLoadIf.Par.MacroList[2].MacroID := 137;

	gMacroLoadIf.Par.MacroList[3].Load := TRUE;
	gMacroLoadIf.Par.MacroList[3].MacroFileName := '138_Circle.xml';
	gMacroLoadIf.Par.MacroList[3].MacroID := 138;

	gMacroLoadIf.Par.MacroList[4].Load := TRUE;
	gMacroLoadIf.Par.MacroList[4].MacroFileName := '180_SpiralProc.xml';
	gMacroLoadIf.Par.MacroList[4].MacroID := 180;

	gMacroLoadIf.Par.MacroList[5].Load := TRUE;
	gMacroLoadIf.Par.MacroList[5].MacroFileName := '139_CircleCCW.xml';
	gMacroLoadIf.Par.MacroList[5].MacroID := 139;

	gMacroLoadIf.Par.MacroList[6].Load := TRUE;
	gMacroLoadIf.Par.MacroList[6].MacroFileName := '140_Sh1Cycle.xml';
	gMacroLoadIf.Par.MacroList[6].MacroID := 140;

	gMacroLoadIf.Par.MacroList[7].Load := TRUE;
	gMacroLoadIf.Par.MacroList[7].MacroFileName := '141_Sh2Cycle.xml';
	gMacroLoadIf.Par.MacroList[7].MacroID := 141;
	//Define the parameters for the macro load IF
	gMacroLoadIf.Par.FileDevice := '6DMacro';
END_PROGRAM
```

### Program Logical/Source/6DCtrl/ProfDemo (IEC)

#### Variables.var
```iecst
VAR
	profFb : ProfBuilderFb;
	moveProf : ProfBuilderParTyp;
	hmiIndex : USINT;
	hmiMove : REFERENCE TO ProfBuilderMoveParTyp;
	resetMove : BOOL;
	state : INT;
	startVibration : BOOL;
	RunMacroFB : MC_BR_MacroRun_Acp6D;
	StopFb : MC_BR_Stop_Acp6D;
	WaitTon : TON;
	shuttleId : USINT;
	vibrationTime : UDINT;
	errorReset : BOOL;
END_VAR
```

#### Cyclic.st
```iecst
(*
	Demo routine

*)

PROGRAM _CYCLIC

	CASE state OF
		0:
			IF startVibration THEN
				RunMacroFB.Controller := ADR(gMcAcp6DController);
				RunMacroFB.ShuttleID := shuttleId;
				RunMacroFB.MacroID := 138;
				RunMacroFB.Execute := TRUE;

				state := 10;
			END_IF
		10:
			IF RunMacroFB.Error THEN
				state := 255;
			ELSIF RunMacroFB.Acknowledge THEN
				RunMacroFB.Execute := FALSE;

				WaitTon.IN := TRUE;
				WaitTon.PT := vibrationTime;

				state := 20;
			END_IF
		20:
			IF WaitTon.Q THEN
				WaitTon.IN := FALSE;
				StopFb.Controller := ADR(gMcAcp6DController);
				StopFb.ShuttleID := shuttleId;
				StopFb.Execute := TRUE;
				state := 30;
			END_IF
		30:
			IF StopFb.Error THEN
				state := 255;
			ELSIF StopFb.Done THEN
				StopFb.Execute := FALSE;
				startVibration := FALSE;

				state := 0;
			END_IF
		255:
			IF errorReset THEN
				StopFb.Execute := FALSE;
				WaitTon.IN := FALSE;
				RunMacroFB.Execute := FALSE;
			END_IF
	END_CASE
	StopFb();
	WaitTon();
	RunMacroFB();

	profFb.Controller := ADR(gMcAcp6DController);
	profFb.Pars := ADR(moveProf);
	profFb();

	IF resetMove THEN
		brsmemset(ADR(hmiMove),0,SIZEOF(moveProf.Moves[0]));
		resetMove := FALSE;
	END_IF

	hmiMove ACCESS ADR(moveProf.Moves[hmiIndex]);

END_PROGRAM
```

### Program Logical/Source/Auxil/Vis (IEC)

#### Types.typ
```iecst
TYPE
	ShVisTyp : 	STRUCT
		ID : USINT;
		Visible : BOOL;
		Color : INT;
		DoseHolder : BOOL;
		CubeHolder : BOOL;
		ProdFill : ARRAY[0..8]OF FillProductTyp;
		ProdColor : INT;
		Pos : McAcp6DShPositionInfoType;
		ScnViewer : ScnViewerConnectionTyp;
	END_STRUCT;
	VisTyp : 	STRUCT
		Shuttles : {REDUND_UNREPLICABLE} ARRAY[0..MAX_SHUTTLE_COUNT_ARRAY]OF ShVisTyp;
		Camera : ARRAY[0..1]OF USINT;
		Robot : RobotTyp;
	END_STRUCT;
	VisShuttleStateEnum :
		(
		VIS_INIT,
		VIS_ACTIVE,
		VIS_ERROR
		);
	ScnViewerConnectionTyp : 	STRUCT
		EnablePositioner : USINT;
		EnablePath : BOOL;
		ClearPath : BOOL;
		PathColor : ARRAY[0..2]OF REAL; (*0-Red, 1-Green, 2-Blue*)
		PathLength : UDINT;
		PathOffset : PointTyp;
	END_STRUCT;
	ShuttleColorEnum :
		(
		COLOR_RED := 1,
		COLOR_BLUE_MATTE,
		COLOR_GREY_MATTE,
		COLOR_YELLOW_MATTE,
		COLOR_GREEN_MATTE,
		COLOR_ORANGE_MATTE,
		COLOR_WHITE_MATTE,
		COLOR_BLACK_MATTE
		);
	PointTyp : 	STRUCT
		X : REAL;
		Y : REAL;
		Z : REAL;
	END_STRUCT;
	RobotTyp : 	STRUCT
		PosQ1 : REAL;
		PosQ2 : REAL;
		PosQ3 : REAL;
		DoseHolder : BOOL;
		CubeHolder : BOOL;
	END_STRUCT;
	FillProductTyp : 	STRUCT
		Vis : BOOL;
		Material : USINT;
	END_STRUCT;
END_TYPE
```

#### Variables.var
```iecst
VAR
	Vis : VisTyp;
	ShData : ARRAY[0..9] OF MC_BR_ShReadPosition_Acp6D;
	states : ARRAY[0..9] OF VisShuttleStateEnum;
	idx : USINT;
	turnOnAllPaths : BOOL;
	clearAllPaths : BOOL;
	i : INT;
END_VAR
```

#### Cyclic.st
```iecst
PROGRAM _CYCLIC
	FOR idx := 0 TO gMainIf.Cfg.ShuttleCount - 1 DO
		IF Vis.Shuttles[idx].ID <> 0 THEN
			Vis.Shuttles[idx].Visible := TRUE;
			Vis.Shuttles[idx].Pos.X := gShuttleIf[idx].Sts.ShuttleInfo.Position.Value.X * 1000;
			Vis.Shuttles[idx].Pos.Y := gShuttleIf[idx].Sts.ShuttleInfo.Position.Value.Y * 1000;
			Vis.Shuttles[idx].Pos.Z := gShuttleIf[idx].Sts.ShuttleInfo.Position.Value.Z * 1000;
			Vis.Shuttles[idx].Pos.RX := gShuttleIf[idx].Sts.ShuttleInfo.Position.Value.RX / 3.14189 * 180.0;
			Vis.Shuttles[idx].Pos.RY := gShuttleIf[idx].Sts.ShuttleInfo.Position.Value.RY / 3.14189 * 180.0;
			Vis.Shuttles[idx].Pos.RZ := gShuttleIf[idx].Sts.ShuttleInfo.Position.Value.RZ / 3.14189 * 180.0;
			CASE gShuttleIf[idx].Sts.ShuttleInfo.State.Value OF
				mcACP6D_SH_STATE_UNDETECTED: (*Shuttle is not detected by the System*)
					Vis.Shuttles[idx].Color := DINT_TO_INT(COLOR_GREY_MATTE);
				mcACP6D_SH_STATE_DISCOVERING: (*Shuttle iis in the process of being discovered by the System		*)
				mcACP6D_SH_STATE_LANDED :  (*Shuttle is landed and controlled by the System. 			*)
					Vis.Shuttles[idx].Color := DINT_TO_INT(COLOR_BLUE_MATTE);
				mcACP6D_SH_STATE_IDLING :  (*Shuttle is levitating and not currently executing a motion command		*)
					Vis.Shuttles[idx].Color := DINT_TO_INT(COLOR_WHITE_MATTE);
				mcACP6D_SH_STATE_DISABLED :  (*Shuttle is not controlled by the System		*)
				mcACP6D_SH_STATE_MOTION :  (*Shuttle is in motion		*)
					Vis.Shuttles[idx].Color := DINT_TO_INT(COLOR_WHITE_MATTE);
				mcACP6D_SH_STATE_WAIT :  (*Shuttle is waiting for a trigger defined by the WaitUntil command		*)
				mcACP6D_SH_STATE_STOPPING :  (*Shuttle is performing an automatic quick stop due to obstacle detection		*)
				mcACP6D_SH_STATE_OBSTACLE :  (*Shuttle is waiting for an obstacle to clear before proceeding*)
					Vis.Shuttles[idx].Color := DINT_TO_INT(COLOR_YELLOW_MATTE);
				mcACP6D_SH_STATE_HOLD :  (*Shuttle is holding position due to positioning error		*)
				mcACP6D_SH_STATE_STOPPED :  (*Shuttle is stopped due to obstacle or boundary detection, it  cannot automatically resume its motion		*)
				mcACP6D_SH_STATE_ERROR :  (*Shuttle has detected an error		*)
					Vis.Shuttles[idx].Color := DINT_TO_INT(COLOR_RED);
				mcACP6D_SH_STATE_RESERVED :  (*Reserved State*)
			END_CASE;
			Vis.Shuttles[idx].ScnViewer.EnablePath := turnOnAllPaths;
			Vis.Shuttles[idx].ScnViewer.ClearPath := clearAllPaths;
		ELSE
			Vis.Shuttles[idx].Visible := TRUE;
		END_IF
	END_FOR;
END_PROGRAM
```

#### Init.st
```iecst
PROGRAM _INIT
	FOR idx := 0 TO gMainIf.Cfg.ShuttleCount - 1 DO
		Vis.Shuttles[idx].ID := idx+1;
		Vis.Shuttles[idx].ScnViewer.PathLength := 35;
	END_FOR;

	Vis.Shuttles[0].ScnViewer.PathColor[0] := 0.0;
	Vis.Shuttles[0].ScnViewer.PathColor[1] := 0.0;
	Vis.Shuttles[0].ScnViewer.PathColor[2] := 0.0;

	Vis.Shuttles[1].ScnViewer.PathColor[0] := 1.0;
	Vis.Shuttles[1].ScnViewer.PathColor[1] := 0.0;
	Vis.Shuttles[1].ScnViewer.PathColor[2] := 0.0;

	Vis.Shuttles[2].ScnViewer.PathColor[0] := 0.0;
	Vis.Shuttles[2].ScnViewer.PathColor[1] := 1.0;
	Vis.Shuttles[2].ScnViewer.PathColor[2] := 0.0;

	Vis.Shuttles[3].ScnViewer.PathColor[0] := 0.0;
	Vis.Shuttles[3].ScnViewer.PathColor[1] := 0.0;
	Vis.Shuttles[3].ScnViewer.PathColor[2] := 1.0;

	Vis.Shuttles[4].ScnViewer.PathColor[0] := 1.0;
	Vis.Shuttles[4].ScnViewer.PathColor[1] := 1.0;
	Vis.Shuttles[4].ScnViewer.PathColor[2] := 0.0;

	Vis.Shuttles[5].ScnViewer.PathColor[0] := 0.75;
	Vis.Shuttles[5].ScnViewer.PathColor[1] := 0.0;
	Vis.Shuttles[5].ScnViewer.PathColor[2] := 0.75;

	Vis.Shuttles[6].ScnViewer.PathColor[0] := 0.0;
	Vis.Shuttles[6].ScnViewer.PathColor[1] := 1.0;
	Vis.Shuttles[6].ScnViewer.PathColor[2] := 1.0;

	Vis.Shuttles[7].ScnViewer.PathColor[0] := 1.0;
	Vis.Shuttles[7].ScnViewer.PathColor[1] := 0.0;
	Vis.Shuttles[7].ScnViewer.PathColor[2] := 0.5;
	turnOnAllPaths := TRUE;
END_PROGRAM
```

### Program Logical/Source/Auxil/Log/LogLib (IEC)

#### Variables.var
```iecst
VAR
	LogServerFb : AsLoggerServer;
END_VAR
```

#### Cyclic.st
```iecst
PROGRAM _CYCLIC
	LogServerFb.port := 15622;
	LogServerFb();

END_PROGRAM
```

- AsLoggerClient.exe (binary file, 27648 bytes)
### Program Logical/Source/Auxil/ProcRecipe (IEC)

#### Types.typ
```iecst
TYPE
	RecipeIfParTyp : 	STRUCT
		FileDevice : STRING[80];
		FileName : STRING[80];
	END_STRUCT;
	RecipeIfCmdTyp : 	STRUCT
		Save : BOOL;
		Load : BOOL;
		Reset : BOOL;
	END_STRUCT;
	RecipeIfStsTyp : 	STRUCT
		Done : USINT;
		Error : USINT;
	END_STRUCT;
	RecipeIfTyp : 	STRUCT
		Cmd : RecipeIfCmdTyp;
		Par : RecipeIfParTyp;
		Sts : RecipeIfStsTyp;
	END_STRUCT;
	RecipeStatesEnum :
		(
		RECIPE_IDLE,
		RECIPE_LOAD,
		RECIPE_SAVE,
		RECIPE_DONE,
		RECIPE_ERROR,
		RECIPE_RESET
		);
END_TYPE
```

#### Variables.var
```iecst
VAR
	recipeXmlFb : MpRecipeXml;
	processRecipeRegParFb : MpRecipeRegPar;
	pickPlaceCfgRegParFb : MpRecipeRegPar;
	pickPlaceTuneRegParFb : MpRecipeRegPar;
	recipeIf : RecipeIfTyp;
	state : RecipeStatesEnum;
END_VAR
```

#### Cyclic.st
```iecst
(*
	Simple program to control the MpRecipe Interface
	Offers ability to save/load recipes on command
*)

PROGRAM _CYCLIC
	CASE state OF
		RECIPE_IDLE: //******************************************************************************** Idle Wait State
			IF recipeXmlFb.Error THEN
				recipeIf.Sts.Error := TRUE;
				state := RECIPE_ERROR;
			ELSIF recipeIf.Cmd.Load THEN
				recipeIf.Cmd.Load := FALSE;
				recipeXmlFb.FileName := ADR(recipeIf.Par.FileName);
				recipeXmlFb.DeviceName := ADR(recipeIf.Par.FileDevice);
				recipeXmlFb.Load := TRUE;
				state := RECIPE_LOAD;
			ELSIF recipeIf.Cmd.Save THEN
				recipeIf.Cmd.Save := FALSE;
				recipeXmlFb.FileName := ADR(recipeIf.Par.FileName);
				recipeXmlFb.DeviceName := ADR(recipeIf.Par.FileDevice);
				recipeXmlFb.Save := TRUE;
				state := RECIPE_SAVE;
			ELSIF recipeIf.Cmd.Reset THEN
			END_IF
		RECIPE_LOAD: //******************************************************************************** Loading recipe state
			IF recipeXmlFb.Error THEN
				state := RECIPE_ERROR;
				recipeIf.Sts.Error := TRUE;
			ELSIF recipeXmlFb.CommandDone THEN
				recipeXmlFb.Load := FALSE;

				recipeIf.Sts.Done := TRUE;
				state := RECIPE_DONE;
			END_IF
		RECIPE_SAVE: //******************************************************************************** Saving recipe state
			IF recipeXmlFb.Error THEN
				state := RECIPE_ERROR;
				recipeIf.Sts.Error := TRUE;
			ELSIF recipeXmlFb.CommandDone THEN
				recipeXmlFb.Save := FALSE;

				recipeIf.Sts.Done := TRUE;
				state := RECIPE_DONE;
			END_IF
		RECIPE_DONE: //******************************************************************************** Done State
			IF NOT recipeIf.Cmd.Load AND NOT recipeIf.Cmd.Save THEN
				state := RECIPE_RESET;
			END_IF
		RECIPE_ERROR: //******************************************************************************** Error State
			IF recipeIf.Cmd.Reset THEN
				recipeXmlFb.ErrorReset := TRUE;
				state := RECIPE_RESET;
			END_IF
		RECIPE_RESET: //******************************************************************************** Reset State
			recipeXmlFb.Save := FALSE;
			recipeXmlFb.Load := FALSE;
			recipeIf.Cmd.Load := FALSE;
			recipeIf.Cmd.Save := FALSE;

			IF NOT recipeXmlFb.Error THEN
				recipeIf.Sts.Done := FALSE;
				recipeIf.Sts.Error := FALSE;

				recipeXmlFb.ErrorReset := FALSE;

				recipeIf.Cmd.Reset := FALSE;

				state := RECIPE_IDLE;
			END_IF
	END_CASE;

	recipeXmlFb();
	processRecipeRegParFb();
	pickPlaceCfgRegParFb();
	pickPlaceTuneRegParFb();
END_PROGRAM
```

#### Exit.st
```iecst
PROGRAM _EXIT
	recipeXmlFb.Enable := FALSE;
	recipeXmlFb();
	processRecipeRegParFb.Enable := FALSE;
	processRecipeRegParFb();
	pickPlaceCfgRegParFb.Enable := FALSE;
	pickPlaceCfgRegParFb();
	pickPlaceTuneRegParFb.Enable := FALSE;
	pickPlaceTuneRegParFb();

END_PROGRAM
```

#### Init.st
```iecst
PROGRAM _INIT

	gProcessRecipe.General.St1St2Cycles := 2;

	gProcessRecipe.Unload.EndPos.X := 0.48;
	gProcessRecipe.Load.EndPos.X := 0.62;

	gProcessRecipe.Inspect.DwellTime := T#1s;
	gProcessRecipe.St1.DwellTime := T#1s;
	gProcessRecipe.St2.DwellTime := T#1s;

	gProcessPickPlaceIf.Par.WaitTune.ApproachHeight := 0;
	gProcessPickPlaceIf.Par.WaitTune.DepartHeight := 00;
	gProcessPickPlaceIf.Par.WaitTune.DwellTime := 0;
	gProcessPickPlaceIf.Par.WaitTune.Radius := 300;

	//Load Parameters and configuration
	gProcessPickPlaceIf.Cfg.LoadPickPos.X := 540;
	gProcessPickPlaceIf.Cfg.LoadPickPos.Y := -60;
	gProcessPickPlaceIf.Cfg.LoadPickPos.Z := 50;

	gProcessPickPlaceIf.Cfg.LoadPlacePos.X := 540;
	gProcessPickPlaceIf.Cfg.LoadPlacePos.Y := 60;
	gProcessPickPlaceIf.Cfg.LoadPlacePos.Z := 40;

	gProcessPickPlaceIf.Par.LoadPickTune.ApproachHeight := 25;
	gProcessPickPlaceIf.Par.LoadPickTune.DepartHeight := 10;
	gProcessPickPlaceIf.Par.LoadPickTune.DwellTime := 75;
	gProcessPickPlaceIf.Par.LoadPickTune.Radius := 10;

	gProcessPickPlaceIf.Par.LoadPlaceTune.ApproachHeight := 30;
	gProcessPickPlaceIf.Par.LoadPlaceTune.DepartHeight := 10;
	gProcessPickPlaceIf.Par.LoadPlaceTune.DwellTime := 50;
	gProcessPickPlaceIf.Par.LoadPlaceTune.Radius := 10;

	//Unload Parameters and configuration
	gProcessPickPlaceIf.Cfg.UnloadPickPos.X := 420;
	gProcessPickPlaceIf.Cfg.UnloadPickPos.Y := 60;
	gProcessPickPlaceIf.Cfg.UnloadPickPos.Z := 40;

	gProcessPickPlaceIf.Cfg.UnloadPlacePos.X := 420;
	gProcessPickPlaceIf.Cfg.UnloadPlacePos.Y := -60;
	gProcessPickPlaceIf.Cfg.UnloadPlacePos.Z := 50;

	gProcessPickPlaceIf.Par.UnloadPickTune.ApproachHeight := 20;
	gProcessPickPlaceIf.Par.UnloadPickTune.DepartHeight := 15;
	gProcessPickPlaceIf.Par.UnloadPickTune.DwellTime := 50;
	gProcessPickPlaceIf.Par.UnloadPickTune.Radius := 25;

	gProcessPickPlaceIf.Par.UnloadPlaceTune.ApproachHeight := 25;
	gProcessPickPlaceIf.Par.UnloadPlaceTune.DepartHeight := 15;
	gProcessPickPlaceIf.Par.UnloadPlaceTune.DwellTime := 75;
	gProcessPickPlaceIf.Par.UnloadPlaceTune.Radius := 5;

	gProcessPickPlaceIf.Par.EmptySpeed.Vel := 1200;
	gProcessPickPlaceIf.Par.EmptySpeed.Accel := 3000;
	gProcessPickPlaceIf.Par.EmptySpeed.Decel := 3000;

	gProcessPickPlaceIf.Par.ProductSpeed.Vel := 700;
	gProcessPickPlaceIf.Par.ProductSpeed.Accel := 3000;
	gProcessPickPlaceIf.Par.ProductSpeed.Decel := 3000;

	gProcessPickPlaceIf.Cfg.WaitPos.X := 420;
	gProcessPickPlaceIf.Cfg.WaitPos.Y := 60;
	gProcessPickPlaceIf.Cfg.WaitPos.Z := 60;

	recipeIf.Par.FileDevice := 'Recipe';
	recipeIf.Par.FileName := 'DemoPars.xml';

	recipeXmlFb.MpLink := ADR(gRecipeXml);
	recipeXmlFb.Enable := TRUE;
	recipeXmlFb.Category := ADR('6D');
	recipeXmlFb();

	processRecipeRegParFb.MpLink := ADR(gRecipeXml);
	processRecipeRegParFb.PVName := ADR('gProcessRecipe');
	processRecipeRegParFb.Enable := TRUE;
	processRecipeRegParFb.Category := ADR('6D');
	processRecipeRegParFb();

	pickPlaceCfgRegParFb.MpLink := ADR(gRecipeXml);
	pickPlaceCfgRegParFb.PVName := ADR('gProcessPickPlaceIf.Cfg');
	pickPlaceCfgRegParFb.Enable := TRUE;
	pickPlaceCfgRegParFb.Category := ADR('6D');
	pickPlaceCfgRegParFb();

	pickPlaceTuneRegParFb.MpLink := ADR(gRecipeXml);
	pickPlaceTuneRegParFb.PVName := ADR('gProcessPickPlaceIf.Par');
	pickPlaceTuneRegParFb.Enable := TRUE;
	pickPlaceTuneRegParFb.Category := ADR('6D');
	pickPlaceTuneRegParFb();
END_PROGRAM
```

### Program Logical/Source/Auxil/Monitor6D (IEC)

#### Types.typ
```iecst
TYPE
	Monitor6DFbsTyp : 	STRUCT
		SegStsFb : ARRAY[0..NUM_SEGMENTS_ARRAY]OF MC_BR_SegGetStatus_Acp6D;
		SysStsFb : MC_BR_SysGetStatus_Acp6D;
		WaitTonFb : TON;
	END_STRUCT;
	Monitor6DStateEnum :
		(
		MON_IDLE,
		MON_SYS_STATUS,
		MON_SEG_STATUS,
		MON_WAIT,
		MON_ERROR,
		MON_RESET
		);
	Monitor6DIfTyp : 	STRUCT
		Cmd : Monitor6DCmdTyp;
		Sts : Monitor6DStsTyp;
	END_STRUCT;
	Monitor6DCmdTyp : 	STRUCT
		DisableMon : BOOL;
		Reset : BOOL;
	END_STRUCT;
	Monitor6DStsTyp : 	STRUCT
		Segments : ARRAY[0..NUM_SEGMENTS_ARRAY]OF McAcp6DGetSegStatusInfoType;
		System : McAcp6DGetSysStatusInfoType;
	END_STRUCT;
END_TYPE
```

#### Variables.var
```iecst
VAR CONSTANT
	NUM_SEGMENTS : USINT := 2;
	NUM_SEGMENTS_ARRAY : USINT := NUM_SEGMENTS-1;
END_VAR
VAR
	state : Monitor6DStateEnum;
	SystemStsIf : Monitor6DIfTyp;
	i : USINT;
	curSegIdx : USINT;
	Fbs : Monitor6DFbsTyp;
	SegStatusCheck : BOOL;
	AbortCount : UDINT;
END_VAR
```

#### Cyclic.st
```iecst
(*
	Task that monitors the 6D system and segment temperatures

	Every Cycle polls a new segment to get it's status, iterates through all segments

	TODO: Will generate an alarm should a any of the segments report a temperature above the configured value

	States
		Wait for 6D system to report available/on
		Check system state
		Check segments temps/status
			Iterates multiplexed through all segments to update the data
		Error
		Reset
*)
PROGRAM _CYCLIC
	CASE state OF
		MON_IDLE:  //******************************************************************************** Idle State
			IF (gAcp6DCtrlIf.Sts.ReadyToPowerOn OR gAcp6DCtrlIf.Sts.PowerOn OR gAcp6DCtrlIf.Sts.Ready) AND NOT SystemStsIf.Cmd.DisableMon THEN
				FOR i:=0 TO NUM_SEGMENTS_ARRAY DO
					Fbs.SegStsFb[i].Controller := ADR(gMcAcp6DController);
					Fbs.SegStsFb[i].SegmentID := i + 1;
				END_FOR;
				Fbs.SysStsFb.Controller := ADR(gMcAcp6DController);
				Fbs.SysStsFb.Execute := TRUE;

				state := MON_SYS_STATUS;
			ELSIF SystemStsIf.Cmd.Reset THEN
				state := MON_RESET;
			END_IF
		MON_SYS_STATUS:  //******************************************************************************** Checking System Status
			IF Fbs.SysStsFb.Error THEN
				state := MON_ERROR;
			ELSIF SystemStsIf.Cmd.DisableMon THEN
				state := MON_RESET;
			ELSIF Fbs.SysStsFb.Valid OR Fbs.SysStsFb.Aborted THEN
				SystemStsIf.Sts.System := Fbs.SysStsFb.SystemInfo;
				Fbs.SysStsFb.Execute := FALSE;

				AbortCount := AbortCount + BOOL_TO_UDINT(Fbs.SysStsFb.Aborted);

				state := MON_SEG_STATUS;
			END_IF
		MON_SEG_STATUS:  //******************************************************************************** Checking the segment status's. Multiplexed
			Fbs.SegStsFb[curSegIdx].Execute := TRUE;
			IF Fbs.SegStsFb[curSegIdx].Error THEN
				state := MON_ERROR;
			ELSIF SystemStsIf.Cmd.DisableMon THEN
				state := MON_RESET;
			ELSIF Fbs.SegStsFb[curSegIdx].Valid OR Fbs.SegStsFb[curSegIdx].Aborted THEN
				Fbs.SegStsFb[curSegIdx].Execute := FALSE;
				SystemStsIf.Sts.Segments[curSegIdx] := Fbs.SegStsFb[curSegIdx].SegmentInfo;
				curSegIdx := curSegIdx + 1;
				AbortCount := AbortCount + BOOL_TO_UDINT(Fbs.SegStsFb[curSegIdx].Aborted);
				IF curSegIdx = NUM_SEGMENTS THEN
					Fbs.WaitTonFb.IN := TRUE;
					Fbs.WaitTonFb.PT := T#5s;
					state := MON_WAIT;
				END_IF
			END_IF
		MON_WAIT:  //******************************************************************************** Wait State
			IF Fbs.WaitTonFb.Q THEN
				Fbs.WaitTonFb.IN := FALSE;

				Fbs.SysStsFb.Execute := TRUE;
				curSegIdx := 0;
				state := MON_SYS_STATUS;
			END_IF
		MON_ERROR:  //******************************************************************************** Error Present State
			state := MON_RESET;
		MON_RESET:  //******************************************************************************** Reset state
			SegStatusCheck := TRUE;
			AbortCount := 0;
			FOR i:=0 TO NUM_SEGMENTS_ARRAY DO
				Fbs.SegStsFb[i].Execute := FALSE;
				SegStatusCheck := Fbs.SegStsFb[i].Error;
			END_FOR;
			Fbs.SysStsFb.Execute := FALSE;
			Fbs.WaitTonFb.IN := FALSE;
			IF SegStatusCheck AND NOT Fbs.SysStsFb.Error THEN
				curSegIdx := 0;
				SystemStsIf.Cmd.Reset := FALSE;

				state := MON_IDLE;
			END_IF
	END_CASE;

	//Fb Calls
	Fbs.SysStsFb();
	Fbs.WaitTonFb();
	FOR i:=0 TO NUM_SEGMENTS_ARRAY DO
		Fbs.SegStsFb[i]();
	END_FOR;
END_PROGRAM
```

#### Init.st
```iecst
PROGRAM _INIT
	//Temporarily disable the monitoring of the status of the system to prevent log book flooding
	SystemStsIf.Cmd.DisableMon := FALSE;

END_PROGRAM
```

### Program Logical/Source/Auxil/SVControl (IEC)

#### Variables.var
```iecst
VAR
	MoveText : STRING[80];
	RadialMove : SV_BE_RadialMove;
	FocalPointMove : SV_BE_FocalPointMove;
	State : State_enum;
	TravelTime : TIME := T#5s;
	Vis : Vis_typ := (Controls:=(TimeInput:=5),Bind:=(FocalPointVisible:=TRUE));
	FocalPointInit : SceneViewCoord_typ := (X:=503,Y:=313,Z:=54);
	StartView : SceneViewCamera_typ := (Perspective:=TRUE,Zoom:=10,Fov:=60.2,ViewPoint:=(X:=1643.43848,Y:=313,Z:=1140),ViewVector:=(X:=-1.14043844,Y:=0,Z:=-1.086),OrientationVector:=(X:=0,Y:=0,Z:=1));
	AngleRad : REAL;
	PointA : SceneViewCamera_typ;
	PointB : SceneViewCamera_typ;
	TotalNumMoves : USINT;
	CompletedMoves : USINT;
	Point : ARRAY[0..2] OF SceneViewCamera_typ;
END_VAR
VAR CONSTANT
	MAX_NUM_MOVES : USINT := 50;
END_VAR
VAR
	MoveNumText : ARRAY[0..MAX_NUM_MOVES] OF STRING[80];
	MoveIndexString : STRING[80];
	IntermediateDateProvider : ARRAY[0..MAX_NUM_MOVES] OF STRING[80];
	DataProvider : ARRAY[0..MAX_NUM_MOVES] OF STRING[80];
	CamMove : ARRAY[0..MAX_NUM_MOVES] OF Move_typ;
	i : USINT;
	FocalPointB : SceneViewCoord_typ;
	FocalPointA : SceneViewCoord_typ;
	SvMovieRecipeFb : MpRecipeXml;
	SvMovieRecipeRegParFb : MpRecipeRegPar;
	svMovieRecipeIf : RecipeCtrlTyp;
	DemoMode : BOOL;
END_VAR
```

#### Main.st
```iecst
PROGRAM _INIT
	(* Insert code here *)

	Point[0] := StartView;
	Vis.Bind.Camera := StartView;

	Vis.Bind.FocalPoint.X := FocalPointInit.X;
	Vis.Bind.FocalPoint.Y := FocalPointInit.Y;
	Vis.Bind.FocalPoint.Z := FocalPointInit.Z;

	Vis.Controls.Linear.X := StartView.ViewPoint.X;
	Vis.Controls.Linear.Y := StartView.ViewPoint.Y;
	Vis.Controls.Z := StartView.ViewPoint.Z;
	Vis.Controls.Fov := StartView.Fov;
	Vis.Controls.Circular.Radius := 100;

	SvMovieRecipeFb.MpLink := ADR(gRecipeSVXml);
	SvMovieRecipeFb.Enable := TRUE;
	SvMovieRecipeFb.Category := ADR('SvMovieCat');
	SvMovieRecipeFb.DeviceName := ADR('SvMovies');
	SvMovieRecipeFb.FileName := ADR(svMovieRecipeIf.Par.FileName);
	svMovieRecipeIf.Par.FileName := 'RadialCamera.xml';
	SvMovieRecipeFb();

	SvMovieRecipeRegParFb.MpLink := ADR(gRecipeSVXml);
	SvMovieRecipeRegParFb.Enable := TRUE;
	SvMovieRecipeRegParFb.Category := ADR('SvMovieCat');
	SvMovieRecipeRegParFb.PVName := ADR('SVControl:CamMove');
	SvMovieRecipeRegParFb();
	svMovieRecipeIf.Cmd.Load := TRUE;

	DemoMode := TRUE;

END_PROGRAM

PROGRAM _CYCLIC
	Vis.Bind.FocalPoint.X := Vis.Bind.FocalPoint.X + Vis.Controls.FocalPoint.XBtnPos - Vis.Controls.FocalPoint.XBtnNeg;
	Vis.Bind.FocalPoint.Y := Vis.Bind.FocalPoint.Y + Vis.Controls.FocalPoint.YBtnPos - Vis.Controls.FocalPoint.YBtnNeg;
	Vis.Bind.FocalPoint.Z := Vis.Bind.FocalPoint.Z + Vis.Controls.FocalPoint.ZBtnPos - Vis.Controls.FocalPoint.ZBtnNeg;

	Vis.Controls.Circular.Radius := Vis.Controls.Circular.Radius + Vis.Controls.Circular.RadiusBtnPos - Vis.Controls.Circular.RadiusBtnNeg;
	Vis.Controls.Linear.X := Vis.Controls.Linear.X + Vis.Controls.Linear.XBtnPos - Vis.Controls.Linear.XBtnNeg;
	Vis.Controls.Linear.Y := Vis.Controls.Linear.Y + Vis.Controls.Linear.YBtnPos - Vis.Controls.Linear.YBtnNeg;

	Vis.Bind.FocalPointVisible := Vis.Controls.FocalPoint.Visible;

	CASE State OF
		MOVE_SETTINGS: //set points
			CASE Vis.Controls.MoveMode OF
				LINEAR:
					MoveText := 'Linear';
					Vis.Bind.Camera.ViewPoint.X := Vis.Controls.Linear.X;
					Vis.Bind.Camera.ViewPoint.Y := Vis.Controls.Linear.Y;

					//keeps view the same when switching to radial mode
					AngleRad := atan2((Vis.Bind.Camera.ViewPoint.Y - Vis.Bind.FocalPoint.Y),(Vis.Bind.Camera.ViewPoint.X - Vis.Bind.FocalPoint.X));
					Vis.Controls.Circular.Angle := AngleRad * 180 / PI;
					IF Vis.Controls.Circular.Angle < 0 THEN
						Vis.Controls.Circular.Angle := Vis.Controls.Circular.Angle + 360;
					ELSIF Vis.Controls.Circular.Angle >= 360 THEN
						Vis.Controls.Circular.Angle := Vis.Controls.Circular.Angle - 360;
					END_IF
					Vis.Controls.Circular.Radius := (Vis.Bind.Camera.ViewPoint.X - Vis.Bind.FocalPoint.X) / COS(AngleRad);
				RADIAL:
					MoveText := 'Radial';
					AngleRad := Vis.Controls.Circular.Angle * PI / 180;

					Vis.Bind.Camera.ViewPoint.X := (Vis.Controls.Circular.Radius * COS(AngleRad)) + Vis.Bind.FocalPoint.X;
					Vis.Bind.Camera.ViewPoint.Y := (Vis.Controls.Circular.Radius * SIN(AngleRad)) + Vis.Bind.FocalPoint.Y;

					Vis.Controls.Linear.X := Vis.Bind.Camera.ViewPoint.X;
					Vis.Controls.Linear.Y := Vis.Bind.Camera.ViewPoint.Y;
			END_CASE

			Vis.Bind.Camera.OrientationVector.X := 0;
			Vis.Bind.Camera.OrientationVector.Y := 0;
			Vis.Bind.Camera.OrientationVector.Z := 1;

			Vis.Bind.Camera.ViewPoint.Z := Vis.Controls.Z;
			Vis.Bind.Camera.Fov := Vis.Controls.Fov;

			Vis.Bind.Camera.ViewVector.X := (Vis.Bind.FocalPoint.X - Vis.Bind.Camera.ViewPoint.X) / 1000.0;
			Vis.Bind.Camera.ViewVector.Y := (Vis.Bind.FocalPoint.Y - Vis.Bind.Camera.ViewPoint.Y) / 1000.0;
			Vis.Bind.Camera.ViewVector.Z := (Vis.Bind.FocalPoint.Z - Vis.Bind.Camera.ViewPoint.Z) / 1000.0;

			IF Vis.Controls.NewMove THEN
				Vis.Controls.NewMove := FALSE;
				State := NEW_MOVE;
			ELSIF Vis.Controls.Load THEN
				State := LOAD_MOVE;
			ELSIF Vis.Controls.Save THEN
				Vis.Controls.Save := FALSE;
				State := SAVE_MOVE;
			END_IF

			IF svMovieRecipeIf.Cmd.Load OR svMovieRecipeIf.Cmd.Save THEN
				SvMovieRecipeFb.Save := svMovieRecipeIf.Cmd.Save;
				SvMovieRecipeFb.Load := svMovieRecipeIf.Cmd.Load;

				State := SAVE_LOAD_RECIPE;
			END_IF

			IF Vis.Controls.SavePointA THEN
				Vis.Controls.SavePointA := FALSE;
				Point[0] := Vis.Bind.Camera;
			END_IF

			IF Vis.Controls.Start OR (DemoMode AND gMainIf.Sts.Running) THEN
				Vis.Controls.Start := TRUE;
				CompletedMoves := 0;
				PointA := Point[0];
				PointB := CamMove[0].Point;
				FocalPointA := FocalPointInit;
				FocalPointB := CamMove[0].FocalPoint;
				State := START_MOVE;
			END_IF

		NEW_MOVE: //new move
			FOR i := 0 TO MAX_NUM_MOVES DO
				IF NOT CamMove[i].IsSaved THEN
					CamMove[i].IsSaved := TRUE;
					CamMove[i].MoveType := Vis.Controls.MoveMode;
					CamMove[i].TravelTime := REAL_TO_TIME(Vis.Controls.TimeInput * 1000);

					State := NEW_MOVE_SAVE;
					EXIT;
				ELSIF i = MAX_NUM_MOVES THEN
					State := MOVE_SETTINGS;
				END_IF
			END_FOR

		NEW_MOVE_SAVE:

			TotalNumMoves := TotalNumMoves + 1;
			CamMove[i].Point := Vis.Bind.Camera;
			CamMove[i].FocalPoint := Vis.Bind.FocalPoint;

			State := UPDATE_LIST;

		UPDATE_LIST:
			brsftoa(i, ADR(MoveIndexString));
			MoveNumText[i] := CONCAT(MoveIndexString, ': ');
			MoveNumText[i] := CONCAT(MoveNumText[i], MoveText);
			MoveNumText[i] := CONCAT(MoveNumText[i], ' Move');

			IntermediateDateProvider[i] := CONCAT('{"value":"',MoveIndexString);
			IntermediateDateProvider[i] := CONCAT(IntermediateDateProvider[i],'","text":"');
			IntermediateDateProvider[i] := CONCAT(IntermediateDateProvider[i], MoveNumText[i]);
			DataProvider[i] := CONCAT(IntermediateDateProvider[i],'"}');

			State := MOVE_SETTINGS;
		SAVE_LOAD_RECIPE:
			IF SvMovieRecipeFb.CommandDone THEN
				IF svMovieRecipeIf.Cmd.Load THEN
					SvMovieRecipeFb.Load := FALSE;
					svMovieRecipeIf.Cmd.Load := FALSE;
					svMovieRecipeIf.Sts.LastLoadedRecipe := svMovieRecipeIf.Par.FileName;

					State := REBUILD_LIST;
				ELSIF svMovieRecipeIf.Cmd.Save THEN
					SvMovieRecipeFb.Save := FALSE;
					svMovieRecipeIf.Cmd.Save := FALSE;

					State := MOVE_SETTINGS;
				END_IF
			END_IF
		REBUILD_LIST:
			brsmemset(ADR(DataProvider),0,SIZEOF(DataProvider));
			brsmemset(ADR(MoveNumText),0,SIZEOF(MoveNumText));
			brsmemset(ADR(IntermediateDateProvider),0,SIZEOF(IntermediateDateProvider));
			TotalNumMoves := 0; //Added for loading saved recipes
			FOR i:=0 TO MAX_NUM_MOVES DO
				IF CamMove[i].IsSaved THEN
					TotalNumMoves := TotalNumMoves + 1;
					brsftoa(i, ADR(MoveIndexString));
					MoveNumText[i] := CONCAT(MoveIndexString, ': ');
					CASE CamMove[i].MoveType OF
						LINEAR:
							MoveNumText[i] := CONCAT(MoveNumText[i], 'Linear');
						RADIAL:
							MoveNumText[i] := CONCAT(MoveNumText[i], 'Radial');
					END_CASE;
					MoveNumText[i] := CONCAT(MoveNumText[i], ' Move');

					IntermediateDateProvider[i] := CONCAT('{"value":"',MoveIndexString);
					IntermediateDateProvider[i] := CONCAT(IntermediateDateProvider[i],'","text":"');
					IntermediateDateProvider[i] := CONCAT(IntermediateDateProvider[i], MoveNumText[i]);
					DataProvider[i] := CONCAT(IntermediateDateProvider[i],'"}');
				END_IF
			END_FOR;

			State := MOVE_SETTINGS;
		LOAD_MOVE: //load
			Vis.Controls.Load := FALSE;

			IF CamMove[Vis.Controls.SelectedMove].IsSaved THEN
				Vis.Controls.Linear.X := CamMove[Vis.Controls.SelectedMove].Point.ViewPoint.X;
				Vis.Controls.Linear.Y := CamMove[Vis.Controls.SelectedMove].Point.ViewPoint.Y;

				Vis.Controls.Z := CamMove[Vis.Controls.SelectedMove].Point.ViewPoint.Z;
				Vis.Controls.Fov := CamMove[Vis.Controls.SelectedMove].Point.Fov;
				Vis.Controls.TimeInput := TIME_TO_REAL(CamMove[Vis.Controls.SelectedMove].TravelTime) / 1000;
				Vis.Controls.MoveMode := CamMove[Vis.Controls.SelectedMove].MoveType;

				Vis.Bind.Camera := CamMove[Vis.Controls.SelectedMove].Point;
				Vis.Bind.FocalPoint := CamMove[Vis.Controls.SelectedMove].FocalPoint;

				//update radial controls
				AngleRad := atan2((Vis.Bind.Camera.ViewPoint.Y - Vis.Bind.FocalPoint.Y),(Vis.Bind.Camera.ViewPoint.X - Vis.Bind.FocalPoint.X));
				Vis.Controls.Circular.Angle := AngleRad * 180 / PI;
				IF Vis.Controls.Circular.Angle < 0 THEN
					Vis.Controls.Circular.Angle := Vis.Controls.Circular.Angle + 360;
				ELSIF Vis.Controls.Circular.Angle >= 360 THEN
					Vis.Controls.Circular.Angle := Vis.Controls.Circular.Angle - 360;
				END_IF
				Vis.Controls.Circular.Radius := (Vis.Bind.Camera.ViewPoint.X - Vis.Bind.FocalPoint.X) / COS(AngleRad);

			END_IF
			State := MOVE_SETTINGS;

		SAVE_MOVE: //save
			IF CamMove[Vis.Controls.SelectedMove].IsSaved THEN
				CamMove[Vis.Controls.SelectedMove].Point := Vis.Bind.Camera;
				CamMove[Vis.Controls.SelectedMove].FocalPoint := Vis.Bind.FocalPoint;
				CamMove[Vis.Controls.SelectedMove].TravelTime := REAL_TO_TIME(Vis.Controls.TimeInput * 1000);
				i := Vis.Controls.SelectedMove;
				State := UPDATE_LIST;
			ELSE
				State := MOVE_SETTINGS;
			END_IF

		START_MOVE:
			TravelTime := CamMove[CompletedMoves].TravelTime;
			IF CamMove[CompletedMoves].MoveType = LINEAR THEN
				State := LINEAR_MOVE;
			ELSIF CamMove[CompletedMoves].MoveType = RADIAL THEN
				State := RADIAL_MOVE;
			END_IF

		RADIAL_MOVE:
			Vis.Controls.SelectedMove := CompletedMoves;
			RadialMove.PointA := PointA;
			RadialMove.PointB := PointB;
			RadialMove.FocalPointA := FocalPointA;
			RadialMove.FocalPointB := FocalPointB;
			RadialMove.TravelTime := TravelTime;
			RadialMove.Execute := TRUE;
			State := WAIT_FOR_RADIAL_MOVE_DONE;

		WAIT_FOR_RADIAL_MOVE_DONE:
			IF RadialMove.Done AND NOT Vis.Controls.Pause THEN
				RadialMove.Execute := FALSE;
				CompletedMoves := CompletedMoves + 1;
				State := MOVE_COMPLETE;
			END_IF

			RadialMove();
			Vis.Controls.ActiveMoveTravelTime := TravelTime;
			Vis.Controls.ActiveMoveElapsedTime := RadialMove.ElapsedTime;
			Vis.Bind.FocalPoint := RadialMove.FocalPointPos;
			Vis.Bind.Camera := RadialMove.SceneViewPos;

		LINEAR_MOVE:
			Vis.Controls.SelectedMove := CompletedMoves;
			FocalPointMove.PointA := PointA;
			FocalPointMove.PointB := PointB;
			//FocalPointMove.FocalPoint := Vis.FocalPoint;
			FocalPointMove.FocalPointA := FocalPointA;
			FocalPointMove.FocalPointB := FocalPointB;
			FocalPointMove.TravelTime := TravelTime;
			FocalPointMove.Execute := TRUE;
			State := WAIT_FOR_LINEAR_MOVE_DONE;

		WAIT_FOR_LINEAR_MOVE_DONE:

			IF FocalPointMove.Done AND NOT Vis.Controls.Pause THEN
				FocalPointMove.Execute := FALSE;
				CompletedMoves := CompletedMoves + 1;
				State := MOVE_COMPLETE;
			END_IF

			FocalPointMove();
			Vis.Controls.ActiveMoveTravelTime := TravelTime;
			Vis.Controls.ActiveMoveElapsedTime := FocalPointMove.ElapsedTime;
			Vis.Bind.FocalPoint := FocalPointMove.FocalPointPos;
			Vis.Bind.Camera := FocalPointMove.SceneViewPos;

		MOVE_COMPLETE:
			IF CompletedMoves < TotalNumMoves THEN
				PointA := Vis.Bind.Camera;
				PointB := CamMove[CompletedMoves].Point;
				FocalPointA := Vis.Bind.FocalPoint;
				FocalPointB := CamMove[CompletedMoves].FocalPoint;
				State := START_MOVE;
			ELSE
				IF DemoMode AND gMainIf.Sts.Running THEN
					Vis.Controls.Start := TRUE;
					CompletedMoves := 0;
					PointA := Point[0];
					PointB := CamMove[0].Point;
					FocalPointA := FocalPointInit;
					FocalPointB := CamMove[0].FocalPoint;
					State := START_MOVE;
				ELSE
					State := WAIT_FOR_STOP;
				END_IF
			END_IF

		WAIT_FOR_STOP:
			IF NOT Vis.Controls.Start THEN
				State := MOVE_SETTINGS;
			END_IF
	END_CASE

	SvMovieRecipeFb();
	SvMovieRecipeRegParFb();

END_PROGRAM

PROGRAM _EXIT
	(* Insert code here *)

END_PROGRAM
```

### Program Logical/Source/ProcessStations/LoadSt (IEC)

#### Types.typ
```iecst
TYPE
	LoadStationStateEnum :
		(
		LOAD_OFF, (*Load station is currently disabled*)
		LOAD_INIT, (*Load station is initalizing*)
		LOAD_WAIT_FOR_SHUTTLE, (*Load Station is waiting for a shuttle*)
		LOAD_WAIT_CFG_IF,
		LOAD_CFG_CYCLIC_POS,
		LOAD_WAIT_ROBOT,
		LOAD_LOADING, (*Load station is loading product onto a shuttle*)
		LOAD_CLEAR_BUFFER,
		LOAD_DONE, (*Load station is done with the unload process*)
		LOAD_ERROR (*Load station had an error*)
		);
	LoadStationFbTyp : 	STRUCT
		Timer : TON;
		ReadCyclicPos : MC_BR_ReadCyclicChAxis_Acp6D;
		RunMacro : MC_BR_MacroRun_Acp6D;
		ClearBuffer : MC_BR_BufferCtrl_Acp6D;
		PathInfluence : MC_BR_OnlinePathInfluence_15;
		Stop : MC_BR_Stop_Acp6D;
		PosGen : MTBasicsLimiter;
	END_STRUCT;
END_TYPE
```

#### Variables.var
```iecst
VAR
	i : INT;
	state : LoadStationStateEnum;
	stationFbs : LoadStationFbTyp;
	stationPars : ProcessRecipeLoadTyp;
	logArgs : ARRAY[0..3] OF UDINT;
	startupCounter : USINT;
END_VAR
```

#### Cyclic.st
```iecst
PROGRAM _CYCLIC

	IF NOT gLoadStIf.Cmd.LocalOverride THEN
		stationPars := gProcessRecipe.Load;
	END_IF

	stationFbs.PosGen.MaxPosSlewRate := gProcessPickPlaceIf.Par.SyncSpeed.Vel;
	stationFbs.PosGen.MaxNegSlewRate := gProcessPickPlaceIf.Par.SyncSpeed.Vel;

	CASE state OF
		LOAD_OFF: //********************************************************************************Load station is currently disabled
			IF gLoadStIf.Cmd.Enable THEN
				startupCounter := 0;
				state := LOAD_INIT;
			ELSIF gLoadStIf.Cmd.Reset THEN
				state := LOAD_ERROR;
			END_IF
		LOAD_INIT: //********************************************************************************Load station is initalizing
			gLoadStIf.Sts.ReadyForNewShuttle := TRUE;
			gLoadStIf.Sts.Enabled := TRUE;

			startupCounter := 0;

			gProcessPickPlaceIf.Par.NextProduct := PROD_DOSING;

			state := LOAD_WAIT_FOR_SHUTTLE;
		LOAD_WAIT_FOR_SHUTTLE: //********************************************************************************Load station is waiting for a shuttle to be present
			//This is a hacky fix to try and fix a SV issue, that's all..
			IF startupCounter < 8 AND NOT gProcessPickPlaceIf.Sts.UnfinishedProductPresent AND gMainIf.Cfg.EnableRobot AND NOT gProcessPickPlaceIf.Cmd.GetLoadPart THEN
				gProcessPickPlaceIf.Sts.RobotProduct := gProcessPickPlaceIf.Par.NextProduct;
			END_IF

			IF NOT gLoadStIf.Cmd.Enable THEN
				gLoadStIf.Sts.ReadyForNewShuttle := FALSE;
				gLoadStIf.Sts.Enabled := FALSE;
				state := LOAD_OFF;
			ELSIF startupCounter < 7 AND NOT gProcessPickPlaceIf.Sts.UnfinishedProductPresent AND gMainIf.Cfg.EnableRobot AND NOT gProcessPickPlaceIf.Cmd.GetLoadPart THEN
				gProcessPickPlaceIf.Cmd.GetLoadPart := TRUE;
				gProcessPickPlaceIf.Sts.RobotProduct := gProcessPickPlaceIf.Par.NextProduct;
			ELSIF gLoadStIf.Par.ShuttleIdx <> STATION_IS_EMPTY AND gLoadStIf.Cmd.Process THEN
				gLoadStIf.Sts.ReadyForNewShuttle := FALSE;
				gLoadStIf.Sts.Processing := TRUE;

				stationFbs.PosGen.Enable := TRUE;
				stationFbs.PosGen.In := 0;
				stationFbs.PosGen.MaxPosSlewRate := gProcessPickPlaceIf.Par.SyncSpeed.Vel;
				stationFbs.PosGen.MaxNegSlewRate := gProcessPickPlaceIf.Par.SyncSpeed.Vel;

				state := LOAD_WAIT_CFG_IF;
			END_IF
		LOAD_WAIT_CFG_IF: //********************************************************************************Waiting for the channel configuration interface to be ready
			IF gCyclicChlCfgIf.Sts.Ready THEN

				gCyclicChlCfgIf.Cmds.Config := TRUE;
				gCyclicChlCfgIf.Pars.LoadShuttleIdx := gLoadStIf.Par.ShuttleIdx;

				state := LOAD_CFG_CYCLIC_POS;
			END_IF
		LOAD_CFG_CYCLIC_POS: //********************************************************************************Waiting for the channel configuration to be configured
			IF gCyclicChlCfgIf.Sts.Ready THEN //Cyclic Channel is configured, we can go ahead and start reading the position
				stationFbs.ReadCyclicPos.Controller := ADR(gMcAcp6DController);
				stationFbs.ReadCyclicPos.ChannelID := 1;
				stationFbs.ReadCyclicPos.AxisID := 1;

				stationFbs.ReadCyclicPos.Enable := TRUE;

				stationFbs.RunMacro.Controller := ADR(gMcAcp6DController);
				stationFbs.RunMacro.MacroID := 150;
				stationFbs.RunMacro.ShuttleID := gShuttleIf[gLoadStIf.Par.ShuttleIdx].Cfg.ShuttleId;
			//	stationFbs.RunMacro.Execute := TRUE;

				logArgs[0] := ADR(gShuttleIf[gLoadStIf.Par.ShuttleIdx].Cfg.ShuttleId);
				logDebug('LoadSt','ShID %d attempted to read CyclicPos and RunLoadMacro',ADR(logArgs));

				state := LOAD_WAIT_ROBOT;
			END_IF
		LOAD_WAIT_ROBOT: //********************************************************************************Waiting for the robot to be ready to load state
			//Waiting for the robot to be ready to pick or alternatively the position value to pass the 'end position'
			IF gDelta.Status.Error THEN
				state := LOAD_ERROR;
			ELSIF gShuttleIf[gLoadStIf.Par.ShuttleIdx].Sts.ShuttleInfo.Position.Value.X >= gProcessRecipe.Load.EndPos.X
					AND stationFbs.ReadCyclicPos.Valid THEN //This should only really happen when we're not using the robot
				logArgs[0] := ADR(gShuttleIf[gLoadStIf.Par.ShuttleIdx].Cfg.ShuttleId);
				logDebug('LoadSt','ShID %d Position passed endpoint with no robot being ready, skipping load.',ADR(logArgs));

				stationFbs.Stop.Controller := ADR(gMcAcp6DController);
				stationFbs.Stop.Execute := TRUE;
				stationFbs.Stop.ShuttleID := gShuttleIf[gLoadStIf.Par.ShuttleIdx].Cfg.ShuttleId;

				state := LOAD_CLEAR_BUFFER;
			ELSIF gProcessPickPlaceIf.Sts.ReadyForLoad AND stationFbs.ReadCyclicPos.Valid AND NOT gProcessPickPlaceIf.Sts.Sync THEN
				logArgs[0] := ADR(gShuttleIf[gLoadStIf.Par.ShuttleIdx].Cfg.ShuttleId);
				logDebug('LoadSt','ShID %d syncing with robot',ADR(logArgs));
				stationFbs.PathInfluence.PositionOffset[0] :=  (stationFbs.ReadCyclicPos.Value) * 1000;
				stationFbs.PathInfluence.AxesGroup := ADR(g3AxDeltaA);
				stationFbs.PathInfluence.CoordSystem := mcMCS;
				stationFbs.PathInfluence.Enable := gProcessPickPlaceIf.Cmd.EnableTracking;

				gProcessPickPlaceIf.Cmd.PickLoad := TRUE;
				gProcessPickPlaceIf.Sts.Sync := TRUE;
				state := LOAD_LOADING;
			END_IF

		LOAD_LOADING: //********************************************************************************Waiting for the load to be complete
			stationFbs.PosGen.In := (stationFbs.ReadCyclicPos.Value - gLoadStIf.Cfg.StationPos.X) * 1000;
			stationFbs.PathInfluence.PositionOffset[0] :=  (stationFbs.ReadCyclicPos.Value) * 1000;

			IF NOT gProcessPickPlaceIf.Sts.UnfinishedProductPresent AND gProcessPickPlaceIf.Sts.Place THEN
				gShuttleIf[gLoadStIf.Par.ShuttleIdx].Sts.ProductState := gProcessPickPlaceIf.Par.NextProduct;
				gProcessPickPlaceIf.Sts.Place := FALSE;
			END_IF

			IF gDelta.Status.Error THEN
				gLoadStIf.Sts.Error := TRUE;
				state := LOAD_ERROR;
			ELSIF NOT gProcessPickPlaceIf.Sts.Sync THEN
				logArgs[0] := ADR(gShuttleIf[gLoadStIf.Par.ShuttleIdx].Cfg.ShuttleId);
				logDebug('LoadSt','ShID %d product removed from robot. Exiting macro movement',ADR(logArgs));

				stationFbs.PosGen.In := 0;

				gProcessPickPlaceIf.Cmd.PickLoad := FALSE;

				stationFbs.Stop.Controller := ADR(gMcAcp6DController);
				stationFbs.Stop.Execute := TRUE;
				stationFbs.Stop.ShuttleID := gShuttleIf[gLoadStIf.Par.ShuttleIdx].Cfg.ShuttleId;

				IF startupCounter <= 7 THEN
					startupCounter := startupCounter + 1;
					gProcessPickPlaceIf.Cmd.GetLoadPart := TRUE;
				END_IF

				IF startupCounter >= 8 AND NOT gUnloadStIf.Sts.Enabled AND NOT gProcessPickPlaceIf.Sts.StartupComplete THEN
					gUnloadStIf.Cmd.Enable := TRUE;
					gProcessPickPlaceIf.Cmd.GetLoadPart := FALSE;
					gProcessPickPlaceIf.Sts.StartupComplete := TRUE;
					gProcessPickPlaceIf.Sts.ReadyForUnload := TRUE;
				END_IF

				state := LOAD_CLEAR_BUFFER;
			END_IF

		LOAD_CLEAR_BUFFER: //********************************************************************************Waiting for the buffer to be cleared
			IF stationFbs.Stop.Error THEN
				logArgs[0] := ADR(stationFbs.ClearBuffer.ErrorID);
				logError('LoadStation','Sh%d had error %d clearing buffer at the load station',ADR(logArgs));
				gLoadStIf.Sts.Error := TRUE;

				state := LOAD_ERROR;
			ELSIF stationFbs.Stop.Done THEN
				stationFbs.RunMacro.Execute := FALSE;
				stationFbs.ReadCyclicPos.Enable := FALSE;
				stationFbs.Stop.Execute := FALSE;

				gShuttleIf[gLoadStIf.Par.ShuttleIdx].Cmd.NextStep := TRUE;

				gLoadStIf.Sts.Processing := FALSE;
				gLoadStIf.Sts.Done := TRUE;

				state := LOAD_DONE;
			END_IF
		LOAD_DONE: //********************************************************************************Load station is done with the load process
			IF NOT gLoadStIf.Cmd.Enable THEN
				gLoadStIf.Sts.Done := FALSE;
				gLoadStIf.Sts.Enabled := FALSE;
				gLoadStIf.Sts.ReadyForNewShuttle := FALSE;
				stationFbs.Timer.IN := FALSE;

				gLoadStIf.Par.ShuttleIdx := STATION_IS_EMPTY;
				state := LOAD_OFF;
			ELSE
				IF gProcessPickPlaceIf.Par.NextProduct = PROD_DOSING THEN
					gProcessPickPlaceIf.Par.NextProduct := PROD_CUBE;
				ELSE
					gProcessPickPlaceIf.Par.NextProduct := PROD_DOSING;
				END_IF

				gLoadStIf.Cmd.Process := FALSE;
				gLoadStIf.Par.ShuttleIdx := STATION_IS_EMPTY;
				gLoadStIf.Sts.Done := FALSE;
				gLoadStIf.Sts.ReadyForNewShuttle := TRUE;

				state := LOAD_WAIT_FOR_SHUTTLE;
			END_IF

		LOAD_ERROR: //********************************************************************************Load station had an error
			IF gLoadStIf.Cmd.Reset THEN
				gLoadStIf.Cmd.Reset := FALSE;

				startupCounter := 0;

				gLoadStIf.Sts.Done := FALSE;
				gLoadStIf.Sts.Enabled := FALSE;
				gLoadStIf.Sts.Error := FALSE;
				gLoadStIf.Sts.Processing := FALSE;
				gLoadStIf.Sts.ReadyForNewShuttle := FALSE;

				stationFbs.RunMacro.Execute := FALSE;
				stationFbs.ReadCyclicPos.Enable := FALSE;
				stationFbs.ClearBuffer.Execute := FALSE;
				stationFbs.Stop.Execute := FALSE;
				stationFbs.Timer.IN := FALSE;
				stationFbs.PathInfluence.Enable := FALSE;

				gLoadStIf.Par.ShuttleIdx := STATION_IS_EMPTY;
				IF gLoadStIf.Cmd.Enable THEN
					state := LOAD_INIT;
				ELSE
					state := LOAD_OFF;
				END_IF
			END_IF
	END_CASE;

	IF NOT gProcessPickPlaceIf.Sts.Sync AND stationFbs.PosGen.Out <= 0.1 AND stationFbs.PosGen.Out >= -0.1 THEN
		stationFbs.PathInfluence.Enable := FALSE;
	END_IF
	stationFbs.PathInfluence.PositionOffset[0] := stationFbs.PosGen.Out;

	stationFbs.RunMacro();
	stationFbs.ReadCyclicPos();
	stationFbs.Stop();
	stationFbs.ClearBuffer();
	stationFbs.PosGen();
	stationFbs.Timer();
	stationFbs.PathInfluence();
END_PROGRAM
```

#### Init.st
```iecst
PROGRAM _INIT
	gLoadStIf.Par.ShuttleIdx := STATION_IS_EMPTY;
	//Define station configuration values
	gLoadStIf.Cfg.StationPos.X := 0.54;
	gLoadStIf.Cfg.StationPos.Y := 0.06;

	stationFbs.PosGen();
END_PROGRAM
```

### Program Logical/Source/ProcessStations/UnloadSt (IEC)

#### Types.typ
```iecst
TYPE
	UnloadStationStateEnum :
		(
		UNLOAD_OFF, (*Unload station is currently disabled*)
		UNLOAD_INIT, (*Unload station is initalizing*)
		UNLOAD_WAIT_FOR_SHUTTLE, (*Unload Station is waiting for a shuttle*)
		UNLOAD_WAIT_CFG_IF,
		UNLOAD_CFG_CYCLIC_POS,
		UNLOAD_WAIT_ROBOT,
		UNLOAD_UNLOADING, (*Unload station is loading product onto a shuttle*)
		UNLOAD_CLEAR_BUFFER,
		UNLOAD_DONE, (*Unload station is done with the unload process*)
		UNLOAD_ERROR (*Unload station had an error*)
		);
	UnloadStationFbTyp : 	STRUCT
		Timer : TON;
		ReadCyclicPos : MC_BR_ReadCyclicChAxis_Acp6D;
		RunMacro : MC_BR_MacroRun_Acp6D;
		ClearBuffer : MC_BR_BufferCtrl_Acp6D;
		PathInfluence : MC_BR_OnlinePathInfluence_15;
		Stop : MC_BR_Stop_Acp6D;
	END_STRUCT;
END_TYPE
```

#### Variables.var
```iecst
VAR
	state : UnloadStationStateEnum;
	stationFbs : UnloadStationFbTyp;
	stationPars : ProcessRecipeLoadTyp;
	logArgs : ARRAY[0..3] OF UDINT;
	productLoadType : BOOL;
END_VAR
```

#### Cyclic.st
```iecst
PROGRAM _CYCLIC

	IF NOT gUnloadStIf.Cmd.LocalOverride THEN
		stationPars := gProcessRecipe.Unload;
	END_IF

	CASE state OF
		UNLOAD_OFF: //********************************************************************************Load station is currently disabled
			IF gUnloadStIf.Cmd.Enable THEN
				state := UNLOAD_INIT;
			ELSIF gUnloadStIf.Cmd.Reset THEN
				state := UNLOAD_ERROR;
			END_IF
		UNLOAD_INIT: //********************************************************************************Load station is initalizing
			gUnloadStIf.Sts.ReadyForNewShuttle := TRUE;
			gUnloadStIf.Sts.Enabled := TRUE;

			state := UNLOAD_WAIT_FOR_SHUTTLE;
		UNLOAD_WAIT_FOR_SHUTTLE: //********************************************************************************Load station is waiting for a shuttle to be present
			IF NOT gUnloadStIf.Cmd.Enable THEN
				gUnloadStIf.Sts.ReadyForNewShuttle := FALSE;
				gUnloadStIf.Sts.Enabled := FALSE;
				state := UNLOAD_OFF;
			ELSIF gUnloadStIf.Par.ShuttleIdx <> STATION_IS_EMPTY AND gUnloadStIf.Cmd.Process THEN
				gUnloadStIf.Sts.ReadyForNewShuttle := FALSE;
				gUnloadStIf.Sts.Processing := TRUE;
				gProcessPickPlaceIf.Sts.RobotProduct := gShuttleIf[gUnloadStIf.Par.ShuttleIdx].Sts.ProductState;

				state := UNLOAD_WAIT_CFG_IF;
			END_IF
		UNLOAD_WAIT_CFG_IF: //********************************************************************************Waiting for the channel configuration interface to be ready
			IF gCyclicChlCfgIf.Sts.Ready THEN
				gCyclicChlCfgIf.Cmds.Config := TRUE;
				gCyclicChlCfgIf.Pars.UnloadShuttleIdx := gUnloadStIf.Par.ShuttleIdx;

				state := UNLOAD_CFG_CYCLIC_POS;
			END_IF
		UNLOAD_CFG_CYCLIC_POS: //********************************************************************************Waiting for the channel configuration to be configured
			IF gCyclicChlCfgIf.Sts.Ready THEN //Cyclic Channel is configured, we can go ahead and start reading the position
				stationFbs.ReadCyclicPos.Controller := ADR(gMcAcp6DController);
				stationFbs.ReadCyclicPos.ChannelID := 2;
				stationFbs.ReadCyclicPos.AxisID := 1;

				stationFbs.ReadCyclicPos.Enable := TRUE;

				stationFbs.RunMacro.Controller := ADR(gMcAcp6DController);
				stationFbs.RunMacro.MacroID := 150;
				stationFbs.RunMacro.ShuttleID := gShuttleIf[gUnloadStIf.Par.ShuttleIdx].Cfg.ShuttleId;
			//	stationFbs.RunMacro.Execute := TRUE;

				logArgs[0] := ADR(gShuttleIf[gUnloadStIf.Par.ShuttleIdx].Cfg.ShuttleId);
				logDebug('UnloadSt','ShID %d attempted to read CyclicPos and RunUnloadMacro',ADR(logArgs));

				state := UNLOAD_WAIT_ROBOT;
			END_IF
		UNLOAD_WAIT_ROBOT: //********************************************************************************Waiting for the robot to be ready to unload state
			//Waiting for the robot to be ready to pick or alternatively the position value to pass the 'end position'
			IF gDelta.Status.Error THEN
				state := UNLOAD_ERROR;
			ELSIF gShuttleIf[gUnloadStIf.Par.ShuttleIdx].Sts.ShuttleInfo.Position.Value.X >= gProcessRecipe.Unload.EndPos.X
					AND stationFbs.ReadCyclicPos.Valid THEN //This should only really happen when we're not using the robot
				logArgs[0] := ADR(gShuttleIf[gUnloadStIf.Par.ShuttleIdx].Cfg.ShuttleId);
				logDebug('UnloadSt','ShID %d Position passed endpoint with no robot being ready, skipping unload.',ADR(logArgs));

				stationFbs.Stop.Controller := ADR(gMcAcp6DController);
				stationFbs.Stop.Execute := TRUE;
				stationFbs.Stop.ShuttleID := gShuttleIf[gUnloadStIf.Par.ShuttleIdx].Cfg.ShuttleId;

				state := UNLOAD_CLEAR_BUFFER;
			ELSIF gProcessPickPlaceIf.Sts.ReadyForUnload AND stationFbs.ReadCyclicPos.Valid AND NOT gProcessPickPlaceIf.Sts.Sync THEN
				logArgs[0] := ADR(gShuttleIf[gUnloadStIf.Par.ShuttleIdx].Cfg.ShuttleId);
				logDebug('UnloadSt','ShID %d syncing with robot',ADR(logArgs));
				stationFbs.PathInfluence.AxesGroup := ADR(g3AxDeltaA);
				stationFbs.PathInfluence.CoordSystem := mcMCS;
				stationFbs.PathInfluence.Enable := gProcessPickPlaceIf.Cmd.EnableTracking;

				gProcessPickPlaceIf.Cmd.PickUnload := TRUE;
				gProcessPickPlaceIf.Sts.Sync := TRUE;
				state := UNLOAD_UNLOADING;
			END_IF

		UNLOAD_UNLOADING: //********************************************************************************Waiting for the unload to be complete
			stationFbs.PathInfluence.PositionOffset[0] := (stationFbs.ReadCyclicPos.Value - gUnloadStIf.Cfg.StationPos.X) * 1000 ;
			IF gDelta.Status.Error THEN
				state := UNLOAD_ERROR;
			ELSIF NOT gProcessPickPlaceIf.Sts.Sync THEN
				logArgs[0] := ADR(gShuttleIf[gUnloadStIf.Par.ShuttleIdx].Cfg.ShuttleId);
				logDebug('UnloadSt','ShID %d product removed from shuttle. Exiting macro movement',ADR(logArgs));

				stationFbs.PathInfluence.Enable := FALSE;
				stationFbs.PathInfluence.PositionOffset[0] := 0;
				gProcessPickPlaceIf.Cmd.PickUnload := FALSE;

				stationFbs.Stop.Controller := ADR(gMcAcp6DController);
				stationFbs.Stop.Execute := TRUE;
				stationFbs.Stop.ShuttleID := gShuttleIf[gUnloadStIf.Par.ShuttleIdx].Cfg.ShuttleId;

				state := UNLOAD_CLEAR_BUFFER;
			END_IF

		UNLOAD_CLEAR_BUFFER: //********************************************************************************Waiting for the buffer to be cleared
			IF stationFbs.Stop.Error THEN
				logArgs[0] := ADR(stationFbs.ClearBuffer.ErrorID);
				logError('UnloadStation','Sh%d had error %d clearing buffer at the unload station',ADR(logArgs));
				gUnloadStIf.Sts.Error := TRUE;

				state := UNLOAD_ERROR;
			ELSIF stationFbs.Stop.Done THEN
				stationFbs.RunMacro.Execute := FALSE;
				stationFbs.ReadCyclicPos.Enable := FALSE;
				stationFbs.Stop.Execute := FALSE;

				gUnloadStIf.Sts.Processing := FALSE;
				gUnloadStIf.Sts.Done := TRUE;
				gShuttleIf[gUnloadStIf.Par.ShuttleIdx].Cmd.NextStep := TRUE;

				state := UNLOAD_DONE;
			END_IF
		UNLOAD_DONE: //********************************************************************************Load station is done with the load process
			IF NOT gUnloadStIf.Cmd.Enable THEN
				gUnloadStIf.Sts.Done := FALSE;
				gUnloadStIf.Sts.Enabled := FALSE;
				gUnloadStIf.Sts.ReadyForNewShuttle := FALSE;
				stationFbs.Timer.IN := FALSE;

				gUnloadStIf.Par.ShuttleIdx := STATION_IS_EMPTY;
				state := UNLOAD_OFF;
			ELSE
				gUnloadStIf.Cmd.Process := FALSE;
				gUnloadStIf.Par.ShuttleIdx := STATION_IS_EMPTY;
				gUnloadStIf.Sts.Done := FALSE;
				gUnloadStIf.Sts.ReadyForNewShuttle := TRUE;

				state := UNLOAD_WAIT_FOR_SHUTTLE;
			END_IF

		UNLOAD_ERROR: //********************************************************************************Load station had an error
			IF gUnloadStIf.Cmd.Reset THEN
				gUnloadStIf.Cmd.Reset := FALSE;

				gUnloadStIf.Sts.Done := FALSE;
				gUnloadStIf.Sts.Enabled := FALSE;
				gUnloadStIf.Sts.Error := FALSE;
				gUnloadStIf.Sts.Processing := FALSE;
				gUnloadStIf.Sts.ReadyForNewShuttle := FALSE;

				stationFbs.RunMacro.Execute := FALSE;
				stationFbs.ReadCyclicPos.Enable := FALSE;
				stationFbs.ClearBuffer.Execute := FALSE;
				stationFbs.Stop.Execute := FALSE;
				stationFbs.Timer.IN := FALSE;
				stationFbs.PathInfluence.Enable := FALSE;

				gUnloadStIf.Par.ShuttleIdx := STATION_IS_EMPTY;
				IF gUnloadStIf.Cmd.Enable THEN
					state := UNLOAD_INIT;
				ELSE
					state := UNLOAD_OFF;
				END_IF
			END_IF
	END_CASE;

	stationFbs.RunMacro();
	stationFbs.ReadCyclicPos();
	stationFbs.ClearBuffer();
	stationFbs.Stop();
	stationFbs.Timer();
	stationFbs.PathInfluence();
END_PROGRAM
```

#### Init.st
```iecst
PROGRAM _INIT
	gUnloadStIf.Par.ShuttleIdx := STATION_IS_EMPTY;
	//Define station configuration values
	gUnloadStIf.Cfg.StationPos.X := 0.42;
	gUnloadStIf.Cfg.StationPos.Y := 0.06;

END_PROGRAM
```

### Program Logical/Source/ProcessStations/ProcessSt (IEC)

#### Cyclic.st - Cyclic code
```iecst
PROGRAM _CYCLIC

	IF NOT pStIf.Cmd.LocalOverride THEN
		stationPars := pStPars;
	END_IF

	CASE state OF
		STATION_OFF: //********************************************************************************Load station is currently disabled
			IF pStIf.Cmd.Enable THEN
				state := STATION_INIT;
			ELSIF pStIf.Cmd.Reset THEN
				state := STATION_ERROR;
			END_IF
		STATION_INIT: //********************************************************************************Load station is initalizing
			pStIf.Sts.ReadyForNewShuttle := TRUE;
			pStIf.Sts.Enabled := TRUE;

			state := STATION_WAIT_FOR_SHUTTLE;
		STATION_WAIT_FOR_SHUTTLE: //********************************************************************************Load station is waiting for a shuttle to be present
			IF NOT pStIf.Cmd.Enable THEN
				pStIf.Sts.ReadyForNewShuttle := FALSE;
				pStIf.Sts.Enabled := FALSE;
				state := STATION_OFF;
			ELSIF pStIf.Par.ShuttleIdx <> STATION_IS_EMPTY AND pStIf.Cmd.Process THEN
				pStIf.Sts.ReadyForNewShuttle := FALSE;
				pStIf.Sts.Processing := TRUE;

				stationFbs.MovePlane.Controller := ADR(gMcAcp6DController);
				stationFbs.MovePlane.Velocity := gProcessRecipe.General.Velocity;
				stationFbs.MovePlane.EndVelocity := 0;
				stationFbs.MovePlane.Acceleration := gProcessRecipe.General.Accel;
				stationFbs.MovePlane.PositionX := stationPars.OperationPos.X;
				stationFbs.MovePlane.PositionY := stationPars.OperationPos.Y;
				stationFbs.MovePlane.Path := mcACP6D_PATH_X_THEN_Y;
				stationFbs.MovePlane.Mode := mcACP6D_MOVE_ABSOLUTE;
				stationFbs.MovePlane.ShuttleID := gShuttleIf[pStIf.Par.ShuttleIdx].Cfg.ShuttleId;
				stationFbs.MovePlane.Execute := TRUE;

				state := STATION_SH_ENTER;
			END_IF
		STATION_SH_ENTER:
			IF stationFbs.MovePlane.Error THEN
				pStIf.Sts.Error := TRUE;
				state := STATION_ERROR;
			ELSIF stationFbs.MovePlane.Done THEN
				stationFbs.MovePlane.Execute := FALSE;

				stationFbs.Timer.IN := TRUE;
				stationFbs.Timer.PT := stationPars.DwellTime;

				CASE gShuttleIf[pStIf.Par.ShuttleIdx].Sts.ProductState OF
					PROD_DOSING:
						IF taskName = 'ProcSt1' THEN
							processDemoTyp := PROC_MATRIX;
						ELSIF taskName = 'ProcSt2' THEN
							processDemoTyp := PROC_SPIRAL;
						END_IF
					PROD_CUBE:
						IF taskName = 'ProcSt1' THEN
							processDemoTyp := PROC_Z_ROT;
						ELSIF taskName = 'ProcSt2' THEN
							processDemoTyp := PROC_NCR;
						END_IF
				END_CASE

				//processDemoTyp := PROC_SPIRAL;
				stationFbs.RunMacroFb.Controller := ADR(gMcAcp6DController);
				stationFbs.RunMacroFb.ShuttleID := gShuttleIf[pStIf.Par.ShuttleIdx].Cfg.ShuttleId;
				CASE processDemoTyp OF
					PROC_SPIRAL:	//************************ Spiral Demo
						stationFbs.RunMacroFb.MacroID := 180;
						stationFbs.RunMacroFb.Execute := TRUE;
					PROC_MATRIX:    //************************ Matrix Demo
						stationFbs.MatrixFb.Controller := ADR(gMcAcp6DController);
						stationFbs.MatrixFb.ShId := gShuttleIf[pStIf.Par.ShuttleIdx].Cfg.ShuttleId;
						stationFbs.MatrixFb.NumColumns := 3;
						stationFbs.MatrixFb.NumRows := 3;
						stationFbs.MatrixFb.FillTime := T#170ms;
						stationFbs.MatrixFb.Velocity := 1;
						stationFbs.MatrixFb.Acceleration := 10;
						stationFbs.MatrixFb.ColSpacing := 0.03;
						stationFbs.MatrixFb.RowSpacing := 0.03;
						stationFbs.MatrixFb.Execute := TRUE;
					PROC_Z_ROT:     //************************ Z Rot Demo
						stationFbs.RunMacroFb.MacroID := 182;
						stationFbs.RunMacroFb.Execute := TRUE;
					PROC_NCR:     //************************ NCR Demo
						stationFbs.NCR_DemoFb.Controller := ADR(gMcAcp6DController);
						stationFbs.NCR_DemoFb.ShId := gShuttleIf[pStIf.Par.ShuttleIdx].Cfg.ShuttleId;
						stationFbs.NCR_DemoFb.Execute := TRUE;
				END_CASE

				state := STATION_OPERATING;
			END_IF

		STATION_OPERATING:
			IF stationFbs.RunMacroFb.Error OR stationFbs.NCR_DemoFb.Error OR stationFbs.MatrixFb.Error THEN
				state := STATION_ERROR;
			ELSIF (stationFbs.RunMacroFb.Execute AND stationFbs.RunMacroFb.Done) OR (stationFbs.NCR_DemoFb.Execute AND stationFbs.NCR_DemoFb.Done) OR (stationFbs.MatrixFb.Execute AND stationFbs.MatrixFb.Done) THEN
				stationFbs.MatrixFb.Execute := FALSE;
				stationFbs.RunMacroFb.Execute := FALSE;
				stationFbs.NCR_DemoFb.Execute := FALSE;
				stationFbs.Timer.IN := FALSE;

				stationFbs.MovePlane.Controller := ADR(gMcAcp6DController);
				stationFbs.MovePlane.Velocity := gProcessRecipe.General.Velocity;
				stationFbs.MovePlane.EndVelocity := 0;
				stationFbs.MovePlane.Acceleration := gProcessRecipe.General.Accel;
				stationFbs.MovePlane.PositionX := stationPars.ExitPos.X;
				stationFbs.MovePlane.PositionY := stationPars.ExitPos.Y;
				stationFbs.MovePlane.Path := mcACP6D_PATH_Y_THEN_X;
				stationFbs.MovePlane.Mode := mcACP6D_MOVE_ABSOLUTE;
				stationFbs.MovePlane.ShuttleID := gShuttleIf[pStIf.Par.ShuttleIdx].Cfg.ShuttleId;
				stationFbs.MovePlane.Execute := TRUE;

				state := STATION_SH_EXIT;
			END_IF

			CASE processDemoTyp OF
				PROC_SPIRAL:
				PROC_MATRIX:
					CASE matrixState OF
						0:
							IF stationFbs.MatrixFb.Filling THEN
								gShuttleIf[pStIf.Par.ShuttleIdx].Sts.ProdFill[stationFbs.MatrixFb.CurrentPocket - 1] := gShuttleIf[pStIf.Par.ShuttleIdx].Sts.ProdFill[stationFbs.MatrixFb.CurrentPocket - 1] + 1;
								matrixState := 1;
							END_IF
						1:
							IF NOT stationFbs.MatrixFb.Filling THEN
								matrixState := 0;
							END_IF
					END_CASE
				PROC_Z_ROT:	//************************ Macro Demos

				PROC_NCR:    //************************ NCR FB Demo
			END_CASE

		STATION_SH_EXIT:
			IF stationFbs.MovePlane.Error THEN
				pStIf.Sts.Error := TRUE;
				state := STATION_ERROR;
			ELSIF stationFbs.MovePlane.Acknowledge THEN
				stationFbs.MovePlane.Execute := FALSE;
				pStIf.Sts.Processing := FALSE;
				pStIf.Sts.Done := TRUE;
				gShuttleIf[pStIf.Par.ShuttleIdx].Cmd.NextStep := TRUE;

				state := STATION_DONE;
			END_IF

		STATION_DONE: //********************************************************************************Load station is done with the load process
			IF NOT pStIf.Cmd.Enable THEN
				pStIf.Sts.Done := FALSE;
				pStIf.Sts.Enabled := FALSE;
				pStIf.Sts.ReadyForNewShuttle := FALSE;
				stationFbs.Timer.IN := FALSE;

				pStIf.Par.ShuttleIdx := STATION_IS_EMPTY;
				state := STATION_OFF;
			ELSE
				pStIf.Cmd.Process := FALSE;
				pStIf.Par.ShuttleIdx := STATION_IS_EMPTY;
				pStIf.Sts.Done := FALSE;
				pStIf.Sts.ReadyForNewShuttle := TRUE;

				state := STATION_WAIT_FOR_SHUTTLE;
			END_IF

		STATION_ERROR: //********************************************************************************Load station had an error
			IF pStIf.Cmd.Reset THEN
				pStIf.Cmd.Reset := FALSE;

				pStIf.Sts.Done := FALSE;
				pStIf.Sts.Enabled := FALSE;
				pStIf.Sts.Error := FALSE;
				pStIf.Sts.Processing := FALSE;
				pStIf.Sts.ReadyForNewShuttle := FALSE;

				stationFbs.Timer.IN := FALSE;
				stationFbs.MovePlane.Execute := FALSE;
				stationFbs.RunMacroFb.Execute := FALSE;
				stationFbs.NCR_DemoFb.Execute := FALSE;
				stationFbs.MatrixFb.Execute := FALSE;

				pStIf.Par.ShuttleIdx := STATION_IS_EMPTY;
				IF pStIf.Cmd.Enable THEN
					state := STATION_INIT;
				ELSE
					state := STATION_OFF;
				END_IF
			END_IF
	END_CASE;

	stationFbs.Timer();
	stationFbs.MovePlane();
	stationFbs.RunMacroFb();
	stationFbs.NCR_DemoFb();
	stationFbs.MatrixFb();
END_PROGRAM
```
